KUKA KRL program: EPS_2_25862_MH5A_A_20251016034302.src

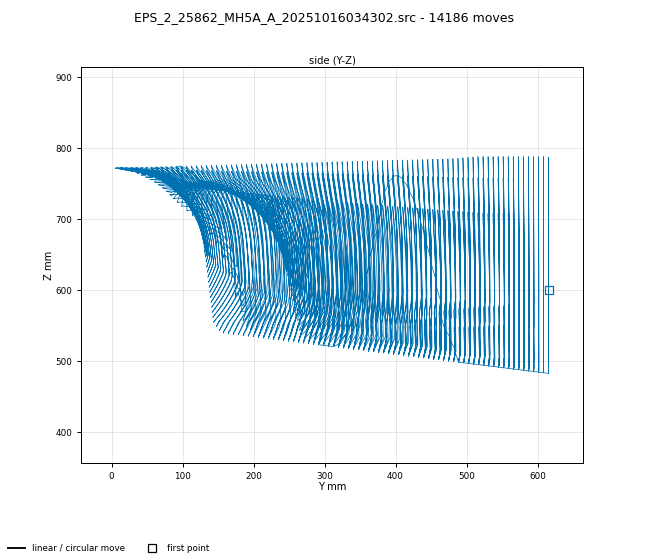
[picture p0: tool path of EPS_2_25862_MH5A_A_20251016034302.src, 14186 of 14188 moves have a stored position in this frame; points joined in program order, loops and branches not executed]
&ACCESS RVP
&REL 4
&COMMENT QRS 19112012
&PARAM EDITMASK = *
DEF PART()
EXT BAS (BAS_COMMAND :IN,REAL :IN )
INT I
BAS (#INITMOV,0 )

;KUKA QRS Post kuka4.cps  Date:22-06-2017 !

File_ID=2891

QRS_PRE_INIT()

;Init var - Until changes are made in qrs_pre_init
Outlet_Square_prg=0
Inlet_1_Square_prg=0
Inlet_2_Square_prg=0
Inlet_3_Square_prg=0
Inlet_4_Square_prg=0
Inlet_5_Square_prg=0

Outlet_1={X 0.000, Y 519.160, Z 687.500, B 0.000, E1 0.000 }
Inlet_1={X 0.000, Y 521.300, Z 657.500, B 0.000, E1 178.000 }
Inlet_2={X 0.000, Y 524.870, Z 607.500, B 0.000, E1 254.000 }
Outlet_1_type=201
Inlet_1_type=201
Inlet_2_type=201
;QRS#1=Sidecore dimensions
;QRS#2=200-8" PVC SDR 35
;QRS#3=200-8" PVC SDR 35
;QRS#4=200-8" PVC SDR 35
;QRS#5=
;QRS#6=
;QRS#7=
;QRS#8=
;QRS#9=12-08 PSX
;QRS#10=12-08 PSX
;QRS#11=12-08 PSX
;QRS#12=
;QRS#13=
;QRS#14=
;QRS#15=
;QRS#16=1220x127x1067 3,5'
;QRS#17=EPS Height
;QRS#18=788
;QRS#19=*
;QRS#20= UPDATED VERSION 22-06-2017
;QRS#21=*
Outlet_Square=0100
Inlet_1_Square=0100
Inlet_2_Square=0100
Inlet_3_Square=0
Inlet_4_Square=0
Inlet_5_Square=0
Mill_Square=1
Outlet_Square_Prg=204
Inlet_1_Square_prg=204
Inlet_2_Square_prg=204

QRS_INIT()

$ADVANCE=5

; T1
PTP {E1 173.595,E2 173.595}
PTP {X 0,Y 615.502,A -85,B 0,C 180,E1 173.595,E2 173.595,E3 0,E4 0,E5 0,E6 0}
QRS_SPEED_INIT()
LIN {X 0,Y 615.502,Z 600,A -85,B 0,C 180,E1 173.595,E2 173.595,E3 0,E4 0,E5 0,E6 0} C_VEL
LIN {X 0,Y 615.502,Z 492.864,A -85,B 0,C 180,E1 173.595,E2 173.595} C_VEL
LIN {X 0,Y 615.502,Z 484.687,A -85,B 0,C 180,E1 173.595,E2 173.595} C_VEL
LIN {X 0,Y 615.49,Z 482.687,A -85,B 0,C 180,E1 173.408,E2 173.408} C_VEL
LIN {X 0,Y 615.493,Z 482.697,A -85,B 0,C 180,E1 170.801,E2 170.801} C_VEL
LIN {X 0,Y 615.479,Z 482.685,A -85,B 0,C 180,E1 168.139,E2 168.139} C_VEL
LIN {X 0,Y 615.488,Z 482.687,A -85,B 0,C 180,E1 165.451,E2 165.451} C_VEL
LIN {X 0,Y 615.492,Z 482.694,A -85,B 0,C 180,E1 162.729,E2 162.729} C_VEL
LIN {X 0,Y 615.477,Z 482.684,A -85,B 0,C 180,E1 159.967,E2 159.967} C_VEL
LIN {X 0,Y 615.494,Z 482.694,A -85,B 0,C 180,E1 157.155,E2 157.155} C_VEL
LIN {X 0,Y 615.493,Z 482.683,A -85,B 0,C 180,E1 154.284,E2 154.284} C_VEL
LIN {X 0,Y 615.484,Z 482.686,A -85,B 0,C 180,E1 151.548,E2 151.548} C_VEL
LIN {X 0,Y 615.491,Z 482.7,A -85,B 0,C 180,E1 148.911,E2 148.911} C_VEL
LIN {X 0,Y 615.479,Z 482.684,A -85,B 0,C 180,E1 145.977,E2 145.977} C_VEL
LIN {X 0,Y 615.481,Z 482.687,A -85,B 0,C 180,E1 143.574,E2 143.574} C_VEL
LIN {X 0,Y 615.495,Z 482.699,A -85,B 0,C 180,E1 140.935,E2 140.935} C_VEL
LIN {X 0,Y 615.488,Z 482.688,A -85,B 0,C 180,E1 138.526,E2 138.526} C_VEL
LIN {X 0,Y 615.477,Z 482.685,A -85,B 0,C 180,E1 135.849,E2 135.849} C_VEL
LIN {X 0,Y 615.496,Z 482.699,A -85,B 0,C 180,E1 133.048,E2 133.048} C_VEL
LIN {X 0,Y 615.489,Z 482.682,A -85,B 0,C 180,E1 130.089,E2 130.089} C_VEL
LIN {X 0,Y 615.492,Z 482.693,A -85,B 0,C 180,E1 127.241,E2 127.241} C_VEL
LIN {X 0,Y 615.485,Z 482.692,A -85,B 0,C 180,E1 124.7,E2 124.7} C_VEL
LIN {X 0,Y 615.49,Z 482.683,A -85,B 0,C 180,E1 122.33,E2 122.33} C_VEL
LIN {X 0,Y 615.476,Z 482.685,A -85,B 0,C 180,E1 119.792,E2 119.792} C_VEL
LIN {X 0,Y 615.498,Z 482.7,A -85,B 0,C 180,E1 117.046,E2 117.046} C_VEL
LIN {X 0,Y 615.489,Z 482.681,A -85,B 0,C 180,E1 114.007,E2 114.007} C_VEL
LIN {X 0,Y 615.474,Z 482.761,A -85,B 0,C 180,E1 113.697,E2 113.697} C_VEL
LIN {X 0,Y 615.484,Z 502.326,A -85,B 0,C 180,E1 110.905,E2 110.905} C_VEL
LIN {X 0,Y 615.489,Z 522.175,A -85,B 0,C 180,E1 108.117,E2 108.117} C_VEL
LIN {X 0,Y 615.494,Z 543.035,A -85,B 0,C 180,E1 105.225,E2 105.225} C_VEL
LIN {X 0,Y 615.481,Z 545.953,A -85,B 0,C 180,E1 104.824,E2 104.824} C_VEL
LIN {X 0,Y 615.48,Z 654.226,A -85,B 0,C 180,E1 103.537,E2 103.537} C_VEL
LIN {X 0,Y 615.487,Z 667.444,A -85,B 0,C 180,E1 103.243,E2 103.243} C_VEL
LIN {X 0,Y 615.487,Z 680.122,A -85,B 0,C 180,E1 102.823,E2 102.823} C_VEL
LIN {X 0,Y 615.487,Z 692.174,A -85,B 0,C 180,E1 102.279,E2 102.279} C_VEL
LIN {X 0,Y 615.49,Z 703.628,A -85,B 0,C 180,E1 101.61,E2 101.61} C_VEL
LIN {X 0,Y 615.496,Z 713.542,A -85,B 0,C 180,E1 100.889,E2 100.889} C_VEL
LIN {X 0,Y 615.497,Z 723.159,A -85,B 0,C 180,E1 100.028,E2 100.028} C_VEL
LIN {X 0,Y 615.496,Z 732.094,A -85,B 0,C 180,E1 99.033,E2 99.033} C_VEL
LIN {X 0,Y 615.499,Z 739.271,A -85,B 0,C 180,E1 98.04,E2 98.04} C_VEL
LIN {X 0,Y 615.496,Z 745.724,A -85,B 0,C 180,E1 96.898,E2 96.898} C_VEL
LIN {X 0,Y 615.497,Z 750.085,A -85,B 0,C 180,E1 95.898,E2 95.898} C_VEL
LIN {X 0,Y 615.498,Z 752.356,A -85,B 0,C 180,E1 95.241,E2 95.241} C_VEL
LIN {X 0,Y 615.496,Z 754.203,A -85,B 0,C 180,E1 94.584,E2 94.584} C_VEL
LIN {X 0,Y 615.496,Z 755.591,A -85,B 0,C 180,E1 93.928,E2 93.928} C_VEL
LIN {X 0,Y 615.495,Z 757.168,A -85,B 0,C 180,E1 92.618,E2 92.618} C_VEL
LIN {X 0,Y 615.5,Z 757.387,A -85,B 0,C 180,E1 91.963,E2 91.963} C_VEL
LIN {X 0,Y 615.495,Z 756.589,A -85,B 0,C 180,E1 90.654,E2 90.654} C_VEL
LIN {X 0,Y 615.497,Z 755.622,A -85,B 0,C 180,E1 90,E2 90} C_VEL
LIN {X 0,Y 615.494,Z 754.255,A -85,B 0,C 180,E1 89.346,E2 89.346} C_VEL
LIN {X 0,Y 615.496,Z 751.382,A -85,B 0,C 180,E1 88.364,E2 88.364} C_VEL
LIN {X 0,Y 615.498,Z 747.492,A -85,B 0,C 180,E1 87.382,E2 87.382} C_VEL
LIN {X 0,Y 615.495,Z 742.483,A -85,B 0,C 180,E1 86.399,E2 86.399} C_VEL
LIN {X 0,Y 615.498,Z 736.194,A -85,B 0,C 180,E1 85.416,E2 85.416} C_VEL
LIN {X 0,Y 615.498,Z 728.32,A -85,B 0,C 180,E1 84.43,E2 84.43} C_VEL
LIN {X 0,Y 615.498,Z 718.54,A -85,B 0,C 180,E1 83.444,E2 83.444} C_VEL
LIN {X 0,Y 615.499,Z 708.271,A -85,B 0,C 180,E1 82.62,E2 82.62} C_VEL
LIN {X 0,Y 615.492,Z 696.728,A -85,B 0,C 180,E1 81.877,E2 81.877} C_VEL
LIN {X 0,Y 615.49,Z 685.198,A -85,B 0,C 180,E1 81.298,E2 81.298} C_VEL
LIN {X 0,Y 615.485,Z 673.274,A -85,B 0,C 180,E1 80.843,E2 80.843} C_VEL
LIN {X 0,Y 615.477,Z 661.229,A -85,B 0,C 180,E1 80.511,E2 80.511} C_VEL
LIN {X 0,Y 615.478,Z 648.035,A -85,B 0,C 180,E1 80.283,E2 80.283} C_VEL
LIN {X 0,Y 615.488,Z 545.884,A -85,B 0,C 180,E1 79.077,E2 79.077} C_VEL
LIN {X 0,Y 615.485,Z 525.776,A -85,B 0,C 180,E1 76.295,E2 76.295} C_VEL
LIN {X 0,Y 615.49,Z 506.326,A -85,B 0,C 180,E1 73.57,E2 73.57} C_VEL
LIN {X 0,Y 615.492,Z 487.095,A -85,B 0,C 180,E1 70.836,E2 70.836} C_VEL
LIN {X 0,Y 615.48,Z 482.686,A -85,B 0,C 180,E1 70.185,E2 70.185} C_VEL
LIN {X 0,Y 615.481,Z 482.685,A -85,B 0,C 180,E1 67.657,E2 67.657} C_VEL
LIN {X 0,Y 615.495,Z 482.699,A -85,B 0,C 180,E1 65.009,E2 65.009} C_VEL
LIN {X 0,Y 615.483,Z 482.683,A -85,B 0,C 180,E1 62.085,E2 62.085} C_VEL
LIN {X 0,Y 615.499,Z 482.68,A -85,B 0,C 180,E1 59.841,E2 59.841} C_VEL
LIN {X 0,Y 615.487,Z 482.687,A -85,B 0,C 180,E1 57.543,E2 57.543} C_VEL
LIN {X 0,Y 615.491,Z 482.697,A -85,B 0,C 180,E1 55.186,E2 55.186} C_VEL
LIN {X 0,Y 615.492,Z 482.691,A -85,B 0,C 180,E1 52.759,E2 52.759} C_VEL
LIN {X 0,Y 615.489,Z 482.682,A -85,B 0,C 180,E1 49.911,E2 49.911} C_VEL
LIN {X 0,Y 615.497,Z 482.694,A -85,B 0,C 180,E1 46.952,E2 46.952} C_VEL
LIN {X 0,Y 615.482,Z 482.684,A -85,B 0,C 180,E1 43.998,E2 43.998} C_VEL
LIN {X 0,Y 615.486,Z 482.7,A -85,B 0,C 180,E1 41.096,E2 41.096} C_VEL
LIN {X 0,Y 615.483,Z 482.693,A -85,B 0,C 180,E1 38.905,E2 38.905} C_VEL
LIN {X 0,Y 615.481,Z 482.684,A -85,B 0,C 180,E1 36.426,E2 36.426} C_VEL
LIN {X 0,Y 615.495,Z 482.691,A -85,B 0,C 180,E1 33.537,E2 33.537} C_VEL
LIN {X 0,Y 615.486,Z 482.884,A -85,B 0,C 180,E1 31.766,E2 31.766} C_VEL
LIN {X 0,Y 615.492,Z 496.948,A -85,B 0,C 180,E1 29.032,E2 29.032} C_VEL
LIN {X 0,Y 615.497,Z 498.159,A -85,B 0,C 180,E1 28.798,E2 28.798} C_VEL
LIN {X 0,Y 615.491,Z 603.751,A -85,B 0,C 180,E1 27.546,E2 27.546} C_VEL
LIN {X 0,Y 615.479,Z 616.47,A -85,B 0,C 180,E1 27.27,E2 27.27} C_VEL
LIN {X 0,Y 615.488,Z 629.197,A -85,B 0,C 180,E1 26.858,E2 26.858} C_VEL
LIN {X 0,Y 615.481,Z 640.719,A -85,B 0,C 180,E1 26.353,E2 26.353} C_VEL
LIN {X 0,Y 615.493,Z 652.002,A -85,B 0,C 180,E1 25.716,E2 25.716} C_VEL
LIN {X 0,Y 615.499,Z 663.389,A -85,B 0,C 180,E1 24.901,E2 24.901} C_VEL
LIN {X 0,Y 615.499,Z 672.008,A -85,B 0,C 180,E1 24.142,E2 24.142} C_VEL
LIN {X 0,Y 615.497,Z 680.725,A -85,B 0,C 180,E1 23.2,E2 23.2} C_VEL
LIN {X 0,Y 615.496,Z 688.627,A -85,B 0,C 180,E1 22.136,E2 22.136} C_VEL
LIN {X 0,Y 615.497,Z 694.828,A -85,B 0,C 180,E1 21.081,E2 21.081} C_VEL
LIN {X 0,Y 615.495,Z 699.584,A -85,B 0,C 180,E1 20.033,E2 20.033} C_VEL
LIN {X 0,Y 615.496,Z 702.046,A -85,B 0,C 180,E1 19.338,E2 19.338} C_VEL
LIN {X 0,Y 615.496,Z 704.133,A -85,B 0,C 180,E1 18.611,E2 18.611} C_VEL
LIN {X 0,Y 615.495,Z 705.544,A -85,B 0,C 180,E1 17.957,E2 17.957} C_VEL
LIN {X 0,Y 615.496,Z 706.572,A -85,B 0,C 180,E1 17.271,E2 17.271} C_VEL
LIN {X 0,Y 615.496,Z 707.28,A -85,B 0,C 180,E1 16.438,E2 16.438} C_VEL
LIN {X 0,Y 615.497,Z 707.12,A -85,B 0,C 180,E1 15.226,E2 15.226} C_VEL
LIN {X 0,Y 615.497,Z 705.525,A -85,B 0,C 180,E1 13.942,E2 13.942} C_VEL
LIN {X 0,Y 615.495,Z 703.871,A -85,B 0,C 180,E1 13.201,E2 13.201} C_VEL
LIN {X 0,Y 615.495,Z 700.772,A -85,B 0,C 180,E1 12.195,E2 12.195} C_VEL
LIN {X 0,Y 615.497,Z 696.609,A -85,B 0,C 180,E1 11.193,E2 11.193} C_VEL
LIN {X 0,Y 615.495,Z 690.251,A -85,B 0,C 180,E1 10.028,E2 10.028} C_VEL
LIN {X 0,Y 615.496,Z 683.344,A -85,B 0,C 180,E1 9.033,E2 9.033} C_VEL
LIN {X 0,Y 615.499,Z 674.712,A -85,B 0,C 180,E1 8.041,E2 8.041} C_VEL
LIN {X 0,Y 615.497,Z 665.894,A -85,B 0,C 180,E1 7.216,E2 7.216} C_VEL
LIN {X 0,Y 615.495,Z 656.246,A -85,B 0,C 180,E1 6.474,E2 6.474} C_VEL
LIN {X 0,Y 615.481,Z 645.657,A -85,B 0,C 180,E1 5.817,E2 5.817} C_VEL
LIN {X 0,Y 615.495,Z 633.852,A -85,B 0,C 180,E1 5.241,E2 5.241} C_VEL
LIN {X 0,Y 615.483,Z 621.635,A -85,B 0,C 180,E1 4.79,E2 4.79} C_VEL
LIN {X 0,Y 615.492,Z 609.025,A -85,B 0,C 180,E1 4.462,E2 4.462} C_VEL
LIN {X 0,Y 615.493,Z 593.991,A -85,B 0,C 180,E1 4.236,E2 4.236} C_VEL
LIN {X 0,Y 615.487,Z 498.146,A -85,B 0,C 180,E1 3.109,E2 3.109} C_VEL
LIN {X 0,Y 615.487,Z 483.823,A -85,B 0,C 180,E1 0.327,E2 0.327} C_VEL
LIN {X 0,Y 615.477,Z 482.689,A -85,B 0,C 180,E1 0.082,E2 0.082} C_VEL
LIN {X 0,Y 615.493,Z 482.682,A -85,B 0,C 180,E1 -2.618,E2 -2.618} C_VEL
LIN {X 0,Y 615.495,Z 482.698,A -85,B 0,C 180,E1 -5.241,E2 -5.241} C_VEL
LIN {X 0,Y 615.479,Z 482.688,A -85,B 0,C 180,E1 -7.876,E2 -7.876} C_VEL
LIN {X 0,Y 615.49,Z 482.683,A -85,B 0,C 180,E1 -10.527,E2 -10.527} C_VEL
LIN {X 0,Y 615.497,Z 482.699,A -85,B 0,C 180,E1 -13.201,E2 -13.201} C_VEL
LIN {X 0,Y 615.48,Z 482.686,A -85,B 0,C 180,E1 -15.905,E2 -15.905} C_VEL
LIN {X 0,Y 615.492,Z 482.685,A -85,B 0,C 180,E1 -18.646,E2 -18.646} C_VEL
LIN {X 0,Y 615.495,Z 482.692,A -85,B 0,C 180,E1 -21.432,E2 -21.432} C_VEL
LIN {X 0,Y 615.478,Z 482.685,A -85,B 0,C 180,E1 -24.272,E2 -24.272} C_VEL
LIN {X 0,Y 615.497,Z 482.698,A -85,B 0,C 180,E1 -27.049,E2 -27.049} C_VEL
LIN {X 0,Y 615.488,Z 482.684,A -85,B 0,C 180,E1 -29.797,E2 -29.797} C_VEL
LIN {X 0,Y 615.484,Z 482.686,A -85,B 0,C 180,E1 -32.458,E2 -32.458} C_VEL
LIN {X 0,Y 615.497,Z 482.692,A -85,B 0,C 180,E1 -34.815,E2 -34.815} C_VEL
LIN {X 0,Y 615.482,Z 482.697,A -85,B 0,C 180,E1 -37.243,E2 -37.243} C_VEL
LIN {X 0,Y 615.498,Z 482.681,A -85,B 0,C 180,E1 -39.749,E2 -39.749} C_VEL
LIN {X 0,Y 615.474,Z 482.688,A -85,B 0,C 180,E1 -42.354,E2 -42.354} C_VEL
LIN {X 0,Y 615.492,Z 482.698,A -85,B 0,C 180,E1 -45.068,E2 -45.068} C_VEL
LIN {X 0,Y 615.488,Z 482.682,A -85,B 0,C 180,E1 -47.92,E2 -47.92} C_VEL
LIN {X 0,Y 615.477,Z 482.687,A -85,B 0,C 180,E1 -50.25,E2 -50.25} C_VEL
LIN {X 0,Y 615.484,Z 482.697,A -85,B 0,C 180,E1 -53.064,E2 -53.064} C_VEL
LIN {X 0,Y 615.487,Z 482.682,A -85,B 0,C 180,E1 -55.979,E2 -55.979} C_VEL
LIN {X 0,Y 615.488,Z 482.7,A -85,B 0,C 180,E1 -58.914,E2 -58.914} C_VEL
LIN {X 0,Y 615.48,Z 482.685,A -85,B 0,C 180,E1 -61.551,E2 -61.551} C_VEL
LIN {X 0,Y 615.477,Z 482.689,A -85,B 0,C 180,E1 -64.284,E2 -64.284} C_VEL
LIN {X 0,Y 615.488,Z 482.751,A -85,B 0,C 180,E1 -66.02,E2 -66.02} C_VEL
LIN {X 0,Y 615.496,Z 506.248,A -85,B 0,C 180,E1 -68.92,E2 -68.92} C_VEL
LIN {X 0,Y 615.483,Z 530.707,A -85,B 0,C 180,E1 -71.881,E2 -71.881} C_VEL
LIN {X 0,Y 615.498,Z 554.974,A -85,B 0,C 180,E1 -74.775,E2 -74.775} C_VEL
LIN {X 0,Y 615.49,Z 574.818,A -85,B 0,C 180,E1 -77.114,E2 -77.114} C_VEL
LIN {X 0,Y 615.477,Z 683.848,A -85,B 0,C 180,E1 -78.411,E2 -78.411} C_VEL
LIN {X 0,Y 615.482,Z 696.355,A -85,B 0,C 180,E1 -78.682,E2 -78.682} C_VEL
LIN {X 0,Y 615.497,Z 709.489,A -85,B 0,C 180,E1 -79.108,E2 -79.108} C_VEL
LIN {X 0,Y 615.48,Z 721.483,A -85,B 0,C 180,E1 -79.64,E2 -79.64} C_VEL
LIN {X 0,Y 615.481,Z 733,A -85,B 0,C 180,E1 -80.304,E2 -80.304} C_VEL
LIN {X 0,Y 615.499,Z 743.344,A -85,B 0,C 180,E1 -81.05,E2 -81.05} C_VEL
LIN {X 0,Y 615.497,Z 751.814,A -85,B 0,C 180,E1 -81.794,E2 -81.794} C_VEL
LIN {X 0,Y 615.498,Z 759.608,A -85,B 0,C 180,E1 -82.62,E2 -82.62} C_VEL
LIN {X 0,Y 615.496,Z 767.204,A -85,B 0,C 180,E1 -83.608,E2 -83.608} C_VEL
LIN {X 0,Y 615.498,Z 774.205,A -85,B 0,C 180,E1 -84.759,E2 -84.759} C_VEL
LIN {X 0,Y 615.493,Z 778.852,A -85,B 0,C 180,E1 -85.744,E2 -85.744} C_VEL
LIN {X 0,Y 615.495,Z 782.399,A -85,B 0,C 180,E1 -86.727,E2 -86.727} C_VEL
LIN {X 0,Y 615.497,Z 784.233,A -85,B 0,C 180,E1 -87.382,E2 -87.382} C_VEL
LIN {X 0,Y 615.496,Z 785.608,A -85,B 0,C 180,E1 -88.037,E2 -88.037} C_VEL
LIN {X 0,Y 615.496,Z 787.174,A -85,B 0,C 180,E1 -89.346,E2 -89.346} C_VEL
LIN {X 0,Y 615.494,Z 787.389,A -85,B 0,C 180,E1 -90,E2 -90} C_VEL
LIN {X 0,Y 615.496,Z 786.58,A -85,B 0,C 180,E1 -91.309,E2 -91.309} C_VEL
LIN {X 0,Y 615.496,Z 785.608,A -85,B 0,C 180,E1 -91.963,E2 -91.963} C_VEL
LIN {X 0,Y 615.497,Z 784.233,A -85,B 0,C 180,E1 -92.618,E2 -92.618} C_VEL
LIN {X 0,Y 615.496,Z 781.35,A -85,B 0,C 180,E1 -93.601,E2 -93.601} C_VEL
LIN {X 0,Y 615.498,Z 777.442,A -85,B 0,C 180,E1 -94.584,E2 -94.584} C_VEL
LIN {X 0,Y 615.499,Z 772.406,A -85,B 0,C 180,E1 -95.57,E2 -95.57} C_VEL
LIN {X 0,Y 615.497,Z 765.869,A -85,B 0,C 180,E1 -96.583,E2 -96.583} C_VEL
LIN {X 0,Y 615.497,Z 758.135,A -85,B 0,C 180,E1 -97.545,E2 -97.545} C_VEL
LIN {X 0,Y 615.498,Z 750.047,A -85,B 0,C 180,E1 -98.371,E2 -98.371} C_VEL
LIN {X 0,Y 615.499,Z 740.17,A -85,B 0,C 180,E1 -99.198,E2 -99.198} C_VEL
LIN {X 0,Y 615.483,Z 728.986,A -85,B 0,C 180,E1 -99.945,E2 -99.945} C_VEL
LIN {X 0,Y 615.481,Z 718.029,A -85,B 0,C 180,E1 -100.527,E2 -100.527} C_VEL
LIN {X 0,Y 615.499,Z 705.423,A -85,B 0,C 180,E1 -101.042,E2 -101.042} C_VEL
LIN {X 0,Y 615.479,Z 693.079,A -85,B 0,C 180,E1 -101.401,E2 -101.401} C_VEL
LIN {X 0,Y 615.477,Z 679.489,A -85,B 0,C 180,E1 -101.652,E2 -101.652} C_VEL
LIN {X 0,Y 615.49,Z 574.818,A -85,B 0,C 180,E1 -102.886,E2 -102.886} C_VEL
LIN {X 0,Y 615.479,Z 550.678,A -85,B 0,C 180,E1 -105.735,E2 -105.735} C_VEL
LIN {X 0,Y 615.493,Z 528.001,A -85,B 0,C 180,E1 -108.444,E2 -108.444} C_VEL
LIN {X 0,Y 615.495,Z 504.813,A -85,B 0,C 180,E1 -111.255,E2 -111.255} C_VEL
LIN {X 0,Y 615.489,Z 482.683,A -85,B 0,C 180,E1 -113.994,E2 -113.994} C_VEL
LIN {X 0,Y 615.48,Z 482.685,A -85,B 0,C 180,E1 -116.444,E2 -116.444} C_VEL
LIN {X 0,Y 615.477,Z 482.689,A -85,B 0,C 180,E1 -118.658,E2 -118.658} C_VEL
LIN {X 0,Y 615.489,Z 482.698,A -85,B 0,C 180,E1 -121.086,E2 -121.086} C_VEL
LIN {X 0,Y 615.487,Z 482.683,A -85,B 0,C 180,E1 -124.021,E2 -124.021} C_VEL
LIN {X 0,Y 615.482,Z 482.695,A -85,B 0,C 180,E1 -126.936,E2 -126.936} C_VEL
LIN {X 0,Y 615.477,Z 482.688,A -85,B 0,C 180,E1 -129.75,E2 -129.75} C_VEL
LIN {X 0,Y 615.49,Z 482.682,A -85,B 0,C 180,E1 -132.351,E2 -132.351} C_VEL
LIN {X 0,Y 615.48,Z 482.7,A -85,B 0,C 180,E1 -135.068,E2 -135.068} C_VEL
LIN {X 0,Y 615.477,Z 482.686,A -85,B 0,C 180,E1 -137.919,E2 -137.919} C_VEL
LIN {X 0,Y 615.498,Z 482.68,A -85,B 0,C 180,E1 -140.251,E2 -140.251} C_VEL
LIN {X 0,Y 615.478,Z 482.701,A -85,B 0,C 180,E1 -143.063,E2 -143.063} C_VEL
LIN {X 0,Y 615.495,Z 482.696,A -85,B 0,C 180,E1 -145.296,E2 -145.296} C_VEL
LIN {X 0,Y 615.485,Z 482.683,A -85,B 0,C 180,E1 -148.314,E2 -148.314} C_VEL
LIN {X 0,Y 615.482,Z 482.687,A -85,B 0,C 180,E1 -150.593,E2 -150.593} C_VEL
LIN {X 0,Y 615.479,Z 482.698,A -85,B 0,C 180,E1 -152.954,E2 -152.954} C_VEL
LIN {X 0,Y 615.478,Z 482.688,A -85,B 0,C 180,E1 -155.728,E2 -155.728} C_VEL
LIN {X 0,Y 615.486,Z 482.686,A -85,B 0,C 180,E1 -158.568,E2 -158.568} C_VEL
LIN {X 0,Y 615.495,Z 482.692,A -85,B 0,C 180,E1 -161.389,E2 -161.389} C_VEL
LIN {X 0,Y 615.48,Z 482.684,A -85,B 0,C 180,E1 -164.095,E2 -164.095} C_VEL
LIN {X 0,Y 615.479,Z 482.693,A -85,B 0,C 180,E1 -166.799,E2 -166.799} C_VEL
LIN {X 0,Y 615.491,Z 482.69,A -85,B 0,C 180,E1 -169.473,E2 -169.473} C_VEL
LIN {X 0,Y 615.479,Z 482.684,A -85,B 0,C 180,E1 -172.124,E2 -172.124} C_VEL
LIN {X 0,Y 615.483,Z 482.692,A -85,B 0,C 180,E1 -174.759,E2 -174.759} C_VEL
LIN {X 0,Y 615.497,Z 482.691,A -85,B 0,C 180,E1 -177.382,E2 -177.382} C_VEL
LIN {X 0,Y 615.477,Z 482.685,A -85,B 0,C 180,E1 -180,E2 -180} C_VEL
LIN {X 0,Y 615.491,Z 482.687,A -85,B 0,C 180,E1 -182.618,E2 -182.618} C_VEL
LIN {X 0,Y 615.493,Z 482.696,A -85,B 0,C 180,E1 -185.241,E2 -185.241} C_VEL
LIN {X 0,Y 615.49,Z 482.687,A -85,B 0,C 180,E1 -186.592,E2 -186.592} C_VEL
LIN {X 0,Y 614.816,Z 482.842,A -85,B 0,C 180,E1 -187.138,E2 -187.138} C_VEL
LIN {X 0,Y 611.984,Z 483.247,A -85,B 0,C 180,E1 -188.024,E2 -188.024} C_VEL
LIN {X 0,Y 609.59,Z 483.561,A -85,B 0,C 180,E1 -188.736,E2 -188.736} C_VEL
LIN {X 0,Y 608.55,Z 483.682,A -85,B 0,C 180,E1 -189.286,E2 -189.286} C_VEL
LIN {X 0,Y 608.459,Z 483.69,A -85,B 0,C 180,E1 -189.472,E2 -189.472} C_VEL
LIN {X 0,Y 608.456,Z 483.687,A -85,B 0,C 180,E1 -192,E2 -192} C_VEL
LIN {X 0,Y 608.476,Z 483.689,A -85,B 0,C 180,E1 -194.721,E2 -194.721} C_VEL
LIN {X 0,Y 608.453,Z 483.691,A -85,B 0,C 180,E1 -197.477,E2 -197.477} C_VEL
LIN {X 0,Y 608.459,Z 483.687,A -85,B 0,C 180,E1 -200.275,E2 -200.275} C_VEL
LIN {X 0,Y 608.455,Z 483.696,A -85,B 0,C 180,E1 -203.124,E2 -203.124} C_VEL
LIN {X 0,Y 608.448,Z 483.688,A -85,B 0,C 180,E1 -206.036,E2 -206.036} C_VEL
LIN {X 0,Y 608.473,Z 483.688,A -85,B 0,C 180,E1 -208.622,E2 -208.622} C_VEL
LIN {X 0,Y 608.474,Z 483.69,A -85,B 0,C 180,E1 -211.316,E2 -211.316} C_VEL
LIN {X 0,Y 608.472,Z 483.686,A -85,B 0,C 180,E1 -213.737,E2 -213.737} C_VEL
LIN {X 0,Y 608.472,Z 483.685,A -85,B 0,C 180,E1 -216.091,E2 -216.091} C_VEL
LIN {X 0,Y 608.472,Z 483.688,A -85,B 0,C 180,E1 -218.588,E2 -218.588} C_VEL
LIN {X 0,Y 608.466,Z 483.691,A -85,B 0,C 180,E1 -221.344,E2 -221.344} C_VEL
LIN {X 0,Y 608.449,Z 483.688,A -85,B 0,C 180,E1 -224.265,E2 -224.265} C_VEL
LIN {X 0,Y 608.462,Z 483.697,A -85,B 0,C 180,E1 -227.042,E2 -227.042} C_VEL
LIN {X 0,Y 608.454,Z 483.688,A -85,B 0,C 180,E1 -229.698,E2 -229.698} C_VEL
LIN {X 0,Y 608.47,Z 483.686,A -85,B 0,C 180,E1 -232.255,E2 -232.255} C_VEL
LIN {X 0,Y 608.452,Z 483.696,A -85,B 0,C 180,E1 -235.095,E2 -235.095} C_VEL
LIN {X 0,Y 608.467,Z 483.685,A -85,B 0,C 180,E1 -237.906,E2 -237.906} C_VEL
LIN {X 0,Y 608.462,Z 483.687,A -85,B 0,C 180,E1 -240.221,E2 -240.221} C_VEL
LIN {X 0,Y 608.485,Z 483.691,A -85,B 0,C 180,E1 -242.793,E2 -242.793} C_VEL
LIN {X 0,Y 608.482,Z 483.684,A -85,B 0,C 180,E1 -245.848,E2 -245.848} C_VEL
LIN {X 0,Y 608.486,Z 483.874,A -85,B 0,C 180,E1 -246.202,E2 -246.202} C_VEL
LIN {X 0,Y 608.541,Z 502.176,A -85,B 0,C 180,E1 -248.845,E2 -248.845} C_VEL
LIN {X 0,Y 608.516,Z 522.072,A -85,B 0,C 180,E1 -251.668,E2 -251.668} C_VEL
LIN {X 0,Y 608.484,Z 543.003,A -85,B 0,C 180,E1 -254.595,E2 -254.595} C_VEL
LIN {X 0,Y 608.468,Z 546.09,A -85,B 0,C 180,E1 -255.023,E2 -255.023} C_VEL
LIN {X 0,Y 608.539,Z 654.234,A -85,B 0,C 180,E1 -256.327,E2 -256.327} C_VEL
LIN {X 0,Y 608.533,Z 667.487,A -85,B 0,C 180,E1 -256.624,E2 -256.624} C_VEL
LIN {X 0,Y 608.513,Z 679.635,A -85,B 0,C 180,E1 -257.027,E2 -257.027} C_VEL
LIN {X 0,Y 608.512,Z 691.904,A -85,B 0,C 180,E1 -257.578,E2 -257.578} C_VEL
LIN {X 0,Y 608.497,Z 703.48,A -85,B 0,C 180,E1 -258.255,E2 -258.255} C_VEL
LIN {X 0,Y 608.481,Z 714.238,A -85,B 0,C 180,E1 -259.042,E2 -259.042} C_VEL
LIN {X 0,Y 608.482,Z 723.247,A -85,B 0,C 180,E1 -259.855,E2 -259.855} C_VEL
LIN {X 0,Y 608.47,Z 732.28,A -85,B 0,C 180,E1 -260.862,E2 -260.862} C_VEL
LIN {X 0,Y 608.464,Z 739.55,A -85,B 0,C 180,E1 -261.866,E2 -261.866} C_VEL
LIN {X 0,Y 608.445,Z 744.449,A -85,B 0,C 180,E1 -262.701,E2 -262.701} C_VEL
LIN {X 0,Y 608.452,Z 748.911,A -85,B 0,C 180,E1 -263.632,E2 -263.632} C_VEL
LIN {X 0,Y 608.442,Z 752.841,A -85,B 0,C 180,E1 -264.698,E2 -264.698} C_VEL
LIN {X 0,Y 608.429,Z 754.719,A -85,B 0,C 180,E1 -265.362,E2 -265.362} C_VEL
LIN {X 0,Y 608.433,Z 756.146,A -85,B 0,C 180,E1 -266.026,E2 -266.026} C_VEL
LIN {X 0,Y 608.421,Z 757.761,A -85,B 0,C 180,E1 -267.352,E2 -267.352} C_VEL
LIN {X 0,Y 608.445,Z 757.998,A -85,B 0,C 180,E1 -268.014,E2 -268.014} C_VEL
LIN {X 0,Y 608.447,Z 757.805,A -85,B 0,C 180,E1 -268.676,E2 -268.676} C_VEL
LIN {X 0,Y 608.437,Z 756.252,A -85,B 0,C 180,E1 -270,E2 -270} C_VEL
LIN {X 0,Y 608.437,Z 754.886,A -85,B 0,C 180,E1 -270.662,E2 -270.662} C_VEL
LIN {X 0,Y 608.44,Z 752.003,A -85,B 0,C 180,E1 -271.655,E2 -271.655} C_VEL
LIN {X 0,Y 608.432,Z 748.099,A -85,B 0,C 180,E1 -272.648,E2 -272.648} C_VEL
LIN {X 0,Y 608.449,Z 743.07,A -85,B 0,C 180,E1 -273.642,E2 -273.642} C_VEL
LIN {X 0,Y 608.465,Z 736.761,A -85,B 0,C 180,E1 -274.637,E2 -274.637} C_VEL
LIN {X 0,Y 608.47,Z 728.87,A -85,B 0,C 180,E1 -275.634,E2 -275.634} C_VEL
LIN {X 0,Y 608.485,Z 719.072,A -85,B 0,C 180,E1 -276.632,E2 -276.632} C_VEL
LIN {X 0,Y 608.479,Z 708.818,A -85,B 0,C 180,E1 -277.466,E2 -277.466} C_VEL
LIN {X 0,Y 608.507,Z 697.295,A -85,B 0,C 180,E1 -278.217,E2 -278.217} C_VEL
LIN {X 0,Y 608.511,Z 685.877,A -85,B 0,C 180,E1 -278.802,E2 -278.802} C_VEL
LIN {X 0,Y 608.533,Z 674.107,A -85,B 0,C 180,E1 -279.263,E2 -279.263} C_VEL
LIN {X 0,Y 608.518,Z 660.533,A -85,B 0,C 180,E1 -279.64,E2 -279.64} C_VEL
LIN {X 0,Y 608.552,Z 648.33,A -85,B 0,C 180,E1 -279.85,E2 -279.85} C_VEL
LIN {X 0,Y 608.476,Z 546.03,A -85,B 0,C 180,E1 -281.075,E2 -281.075} C_VEL
LIN {X 0,Y 608.5,Z 525.828,A -85,B 0,C 180,E1 -283.894,E2 -283.894} C_VEL
LIN {X 0,Y 608.511,Z 507.114,A -85,B 0,C 180,E1 -286.541,E2 -286.541} C_VEL
LIN {X 0,Y 608.556,Z 488.485,A -85,B 0,C 180,E1 -289.216,E2 -289.216} C_VEL
LIN {X 0,Y 608.457,Z 483.689,A -85,B 0,C 180,E1 -289.921,E2 -289.921} C_VEL
LIN {X 0,Y 608.463,Z 483.688,A -85,B 0,C 180,E1 -292.476,E2 -292.476} C_VEL
LIN {X 0,Y 608.458,Z 483.69,A -85,B 0,C 180,E1 -294.57,E2 -294.57} C_VEL
LIN {X 0,Y 608.486,Z 483.691,A -85,B 0,C 180,E1 -297.207,E2 -297.207} C_VEL
LIN {X 0,Y 608.465,Z 483.686,A -85,B 0,C 180,E1 -299.97,E2 -299.97} C_VEL
LIN {X 0,Y 608.462,Z 483.689,A -85,B 0,C 180,E1 -302.522,E2 -302.522} C_VEL
LIN {X 0,Y 608.439,Z 483.694,A -85,B 0,C 180,E1 -305.277,E2 -305.277} C_VEL
LIN {X 0,Y 608.47,Z 483.685,A -85,B 0,C 180,E1 -307.745,E2 -307.745} C_VEL
LIN {X 0,Y 608.455,Z 483.689,A -85,B 0,C 180,E1 -310.329,E2 -310.329} C_VEL
LIN {X 0,Y 608.485,Z 483.687,A -85,B 0,C 180,E1 -313.31,E2 -313.31} C_VEL
LIN {X 0,Y 608.469,Z 483.686,A -85,B 0,C 180,E1 -316.13,E2 -316.13} C_VEL
LIN {X 0,Y 608.457,Z 483.698,A -85,B 0,C 180,E1 -318.823,E2 -318.823} C_VEL
LIN {X 0,Y 608.465,Z 483.687,A -85,B 0,C 180,E1 -321.411,E2 -321.411} C_VEL
LIN {X 0,Y 608.472,Z 483.685,A -85,B 0,C 180,E1 -323.949,E2 -323.949} C_VEL
LIN {X 0,Y 608.467,Z 483.689,A -85,B 0,C 180,E1 -326.329,E2 -326.329} C_VEL
LIN {X 0,Y 608.47,Z 483.805,A -85,B 0,C 180,E1 -328.198,E2 -328.198} C_VEL
LIN {X 0,Y 608.469,Z 498.316,A -85,B 0,C 180,E1 -331.038,E2 -331.038} C_VEL
LIN {X 0,Y 608.588,Z 508.378,A -85,B 0,C 180,E1 -331.176,E2 -331.176} C_VEL
LIN {X 0,Y 608.538,Z 604.65,A -85,B 0,C 180,E1 -332.334,E2 -332.334} C_VEL
LIN {X 0,Y 608.519,Z 618.171,A -85,B 0,C 180,E1 -332.643,E2 -332.643} C_VEL
LIN {X 0,Y 608.526,Z 630.922,A -85,B 0,C 180,E1 -333.077,E2 -333.077} C_VEL
LIN {X 0,Y 608.506,Z 642.266,A -85,B 0,C 180,E1 -333.598,E2 -333.598} C_VEL
LIN {X 0,Y 608.481,Z 653.778,A -85,B 0,C 180,E1 -334.274,E2 -334.274} C_VEL
LIN {X 0,Y 608.483,Z 664.536,A -85,B 0,C 180,E1 -335.066,E2 -335.066} C_VEL
LIN {X 0,Y 608.465,Z 674.673,A -85,B 0,C 180,E1 -336.002,E2 -336.002} C_VEL
LIN {X 0,Y 608.469,Z 682.396,A -85,B 0,C 180,E1 -336.876,E2 -336.876} C_VEL
LIN {X 0,Y 608.454,Z 690.095,A -85,B 0,C 180,E1 -337.951,E2 -337.951} C_VEL
LIN {X 0,Y 608.431,Z 696.085,A -85,B 0,C 180,E1 -339.017,E2 -339.017} C_VEL
LIN {X 0,Y 608.434,Z 700.699,A -85,B 0,C 180,E1 -340.077,E2 -340.077} C_VEL
LIN {X 0,Y 608.425,Z 704.533,A -85,B 0,C 180,E1 -341.293,E2 -341.293} C_VEL
LIN {X 0,Y 608.42,Z 706.949,A -85,B 0,C 180,E1 -342.522,E2 -342.522} C_VEL
LIN {X 0,Y 608.422,Z 707.851,A -85,B 0,C 180,E1 -343.481,E2 -343.481} C_VEL
LIN {X 0,Y 608.42,Z 707.863,A -85,B 0,C 180,E1 -344.592,E2 -344.592} C_VEL
LIN {X 0,Y 608.418,Z 707.29,A -85,B 0,C 180,E1 -345.278,E2 -345.278} C_VEL
LIN {X 0,Y 608.431,Z 706.267,A -85,B 0,C 180,E1 -345.992,E2 -345.992} C_VEL
LIN {X 0,Y 608.437,Z 704.93,A -85,B 0,C 180,E1 -346.643,E2 -346.643} C_VEL
LIN {X 0,Y 608.431,Z 701.982,A -85,B 0,C 180,E1 -347.661,E2 -347.661} C_VEL
LIN {X 0,Y 608.452,Z 697.98,A -85,B 0,C 180,E1 -348.676,E2 -348.676} C_VEL
LIN {X 0,Y 608.443,Z 691.825,A -85,B 0,C 180,E1 -349.854,E2 -349.854} C_VEL
LIN {X 0,Y 608.469,Z 685.104,A -85,B 0,C 180,E1 -350.862,E2 -350.862} C_VEL
LIN {X 0,Y 608.462,Z 676.803,A -85,B 0,C 180,E1 -351.866,E2 -351.866} C_VEL
LIN {X 0,Y 608.49,Z 668.305,A -85,B 0,C 180,E1 -352.701,E2 -352.701} C_VEL
LIN {X 0,Y 608.476,Z 657.879,A -85,B 0,C 180,E1 -353.534,E2 -353.534} C_VEL
LIN {X 0,Y 608.483,Z 647.596,A -85,B 0,C 180,E1 -354.199,E2 -354.199} C_VEL
LIN {X 0,Y 608.526,Z 636.324,A -85,B 0,C 180,E1 -354.782,E2 -354.782} C_VEL
LIN {X 0,Y 608.526,Z 624.862,A -85,B 0,C 180,E1 -355.238,E2 -355.238} C_VEL
LIN {X 0,Y 608.55,Z 611.74,A -85,B 0,C 180,E1 -355.612,E2 -355.612} C_VEL
LIN {X 0,Y 608.552,Z 599.021,A -85,B 0,C 180,E1 -355.84,E2 -355.84} C_VEL
LIN {X 0,Y 608.449,Z 498.372,A -85,B 0,C 180,E1 -357.041,E2 -357.041} C_VEL
LIN {X 0,Y 608.451,Z 484.1,A -85,B 0,C 180,E1 -359.834,E2 -359.834} C_VEL
LIN {X 0,Y 608.467,Z 483.687,A -85,B 0,C 180,E1 -360,E2 -360} C_VEL
LIN {X 0,Y 608.482,Z 483.685,A -85,B 0,C 180,E1 -362.648,E2 -362.648} C_VEL
LIN {X 0,Y 608.471,Z 483.696,A -85,B 0,C 180,E1 -365.302,E2 -365.302} C_VEL
LIN {X 0,Y 608.471,Z 483.686,A -85,B 0,C 180,E1 -367.967,E2 -367.967} C_VEL
LIN {X 0,Y 608.467,Z 483.687,A -85,B 0,C 180,E1 -370.65,E2 -370.65} C_VEL
LIN {X 0,Y 608.469,Z 483.694,A -85,B 0,C 180,E1 -373.356,E2 -373.356} C_VEL
LIN {X 0,Y 608.455,Z 483.687,A -85,B 0,C 180,E1 -376.094,E2 -376.094} C_VEL
LIN {X 0,Y 608.456,Z 483.692,A -85,B 0,C 180,E1 -378.87,E2 -378.87} C_VEL
LIN {X 0,Y 608.47,Z 483.688,A -85,B 0,C 180,E1 -381.691,E2 -381.691} C_VEL
LIN {X 0,Y 608.451,Z 483.689,A -85,B 0,C 180,E1 -384.571,E2 -384.571} C_VEL
LIN {X 0,Y 608.482,Z 483.693,A -85,B 0,C 180,E1 -387.211,E2 -387.211} C_VEL
LIN {X 0,Y 608.464,Z 483.686,A -85,B 0,C 180,E1 -389.973,E2 -389.973} C_VEL
LIN {X 0,Y 608.458,Z 483.689,A -85,B 0,C 180,E1 -392.524,E2 -392.524} C_VEL
LIN {X 0,Y 608.453,Z 483.694,A -85,B 0,C 180,E1 -395.277,E2 -395.277} C_VEL
LIN {X 0,Y 608.464,Z 483.687,A -85,B 0,C 180,E1 -397.747,E2 -397.747} C_VEL
LIN {X 0,Y 608.447,Z 483.689,A -85,B 0,C 180,E1 -400.33,E2 -400.33} C_VEL
LIN {X 0,Y 608.465,Z 483.691,A -85,B 0,C 180,E1 -403.31,E2 -403.31} C_VEL
LIN {X 0,Y 608.469,Z 483.686,A -85,B 0,C 180,E1 -406.132,E2 -406.132} C_VEL
LIN {X 0,Y 608.455,Z 483.696,A -85,B 0,C 180,E1 -408.825,E2 -408.825} C_VEL
LIN {X 0,Y 608.466,Z 483.688,A -85,B 0,C 180,E1 -411.413,E2 -411.413} C_VEL
LIN {X 0,Y 608.457,Z 483.687,A -85,B 0,C 180,E1 -413.953,E2 -413.953} C_VEL
LIN {X 0,Y 608.463,Z 483.688,A -85,B 0,C 180,E1 -416.33,E2 -416.33} C_VEL
LIN {X 0,Y 608.476,Z 483.693,A -85,B 0,C 180,E1 -418.728,E2 -418.728} C_VEL
LIN {X 0,Y 608.466,Z 483.688,A -85,B 0,C 180,E1 -421.382,E2 -421.382} C_VEL
LIN {X 0,Y 608.438,Z 483.69,A -85,B 0,C 180,E1 -423.965,E2 -423.965} C_VEL
LIN {X 0,Y 608.482,Z 483.708,A -85,B 0,C 180,E1 -425.847,E2 -425.847} C_VEL
LIN {X 0,Y 608.609,Z 499.073,A -85,B 0,C 180,E1 -427.779,E2 -427.779} C_VEL
LIN {X 0,Y 608.544,Z 522.033,A -85,B 0,C 180,E1 -430.608,E2 -430.608} C_VEL
LIN {X 0,Y 608.525,Z 543.558,A -85,B 0,C 180,E1 -433.218,E2 -433.218} C_VEL
LIN {X 0,Y 608.504,Z 566.578,A -85,B 0,C 180,E1 -435.971,E2 -435.971} C_VEL
LIN {X 0,Y 608.524,Z 575.275,A -85,B 0,C 180,E1 -436.974,E2 -436.974} C_VEL
LIN {X 0,Y 608.534,Z 683.962,A -85,B 0,C 180,E1 -438.277,E2 -438.277} C_VEL
LIN {X 0,Y 608.533,Z 697.225,A -85,B 0,C 180,E1 -438.572,E2 -438.572} C_VEL
LIN {X 0,Y 608.544,Z 710.333,A -85,B 0,C 180,E1 -439.009,E2 -439.009} C_VEL
LIN {X 0,Y 608.498,Z 721.64,A -85,B 0,C 180,E1 -439.519,E2 -439.519} C_VEL
LIN {X 0,Y 608.471,Z 733.201,A -85,B 0,C 180,E1 -440.191,E2 -440.191} C_VEL
LIN {X 0,Y 608.485,Z 743.596,A -85,B 0,C 180,E1 -440.946,E2 -440.946} C_VEL
LIN {X 0,Y 608.475,Z 752.114,A -85,B 0,C 180,E1 -441.699,E2 -441.699} C_VEL
LIN {X 0,Y 608.471,Z 759.962,A -85,B 0,C 180,E1 -442.534,E2 -442.534} C_VEL
LIN {X 0,Y 608.46,Z 767.287,A -85,B 0,C 180,E1 -443.485,E2 -443.485} C_VEL
LIN {X 0,Y 608.45,Z 772.867,A -85,B 0,C 180,E1 -444.366,E2 -444.366} C_VEL
LIN {X 0,Y 608.432,Z 777.951,A -85,B 0,C 180,E1 -445.362,E2 -445.362} C_VEL
LIN {X 0,Y 608.449,Z 781.896,A -85,B 0,C 180,E1 -446.358,E2 -446.358} C_VEL
LIN {X 0,Y 608.425,Z 784.809,A -85,B 0,C 180,E1 -447.352,E2 -447.352} C_VEL
LIN {X 0,Y 608.441,Z 786.201,A -85,B 0,C 180,E1 -448.014,E2 -448.014} C_VEL
LIN {X 0,Y 608.438,Z 787.783,A -85,B 0,C 180,E1 -449.338,E2 -449.338} C_VEL
LIN {X 0,Y 608.434,Z 788,A -85,B 0,C 180,E1 -450,E2 -450} C_VEL
LIN {X 0,Y 608.448,Z 787.184,A -85,B 0,C 180,E1 -451.324,E2 -451.324} C_VEL
LIN {X 0,Y 608.441,Z 786.201,A -85,B 0,C 180,E1 -451.986,E2 -451.986} C_VEL
LIN {X 0,Y 608.425,Z 784.809,A -85,B 0,C 180,E1 -452.648,E2 -452.648} C_VEL
LIN {X 0,Y 608.449,Z 781.896,A -85,B 0,C 180,E1 -453.642,E2 -453.642} C_VEL
LIN {X 0,Y 608.432,Z 777.951,A -85,B 0,C 180,E1 -454.638,E2 -454.638} C_VEL
LIN {X 0,Y 608.437,Z 771.877,A -85,B 0,C 180,E1 -455.801,E2 -455.801} C_VEL
LIN {X 0,Y 608.462,Z 765.236,A -85,B 0,C 180,E1 -456.799,E2 -456.799} C_VEL
LIN {X 0,Y 608.455,Z 756.991,A -85,B 0,C 180,E1 -457.8,E2 -457.8} C_VEL
LIN {X 0,Y 608.472,Z 748.539,A -85,B 0,C 180,E1 -458.636,E2 -458.636} C_VEL
LIN {X 0,Y 608.474,Z 738.094,A -85,B 0,C 180,E1 -459.473,E2 -459.473} C_VEL
LIN {X 0,Y 608.482,Z 727.76,A -85,B 0,C 180,E1 -460.145,E2 -460.145} C_VEL
LIN {X 0,Y 608.521,Z 716.245,A -85,B 0,C 180,E1 -460.741,E2 -460.741} C_VEL
LIN {X 0,Y 608.528,Z 704.883,A -85,B 0,C 180,E1 -461.192,E2 -461.192} C_VEL
LIN {X 0,Y 608.535,Z 692.28,A -85,B 0,C 180,E1 -461.554,E2 -461.554} C_VEL
LIN {X 0,Y 608.535,Z 679.622,A -85,B 0,C 180,E1 -461.787,E2 -461.787} C_VEL
LIN {X 0,Y 608.489,Z 574.948,A -85,B 0,C 180,E1 -463.037,E2 -463.037} C_VEL
LIN {X 0,Y 608.512,Z 550.733,A -85,B 0,C 180,E1 -465.92,E2 -465.92} C_VEL
LIN {X 0,Y 608.566,Z 526.338,A -85,B 0,C 180,E1 -468.866,E2 -468.866} C_VEL
LIN {X 0,Y 608.589,Z 503.378,A -85,B 0,C 180,E1 -471.687,E2 -471.687} C_VEL
LIN {X 0,Y 608.603,Z 484.346,A -85,B 0,C 180,E1 -474.067,E2 -474.067} C_VEL
LIN {X 0,Y 608.469,Z 483.687,A -85,B 0,C 180,E1 -474.197,E2 -474.197} C_VEL
LIN {X 0,Y 608.481,Z 483.695,A -85,B 0,C 180,E1 -477.207,E2 -477.207} C_VEL
LIN {X 0,Y 608.466,Z 483.686,A -85,B 0,C 180,E1 -479.971,E2 -479.971} C_VEL
LIN {X 0,Y 608.457,Z 483.688,A -85,B 0,C 180,E1 -482.521,E2 -482.521} C_VEL
LIN {X 0,Y 608.434,Z 483.699,A -85,B 0,C 180,E1 -485.277,E2 -485.277} C_VEL
LIN {X 0,Y 608.47,Z 483.687,A -85,B 0,C 180,E1 -487.745,E2 -487.745} C_VEL
LIN {X 0,Y 608.45,Z 483.688,A -85,B 0,C 180,E1 -490.329,E2 -490.329} C_VEL
LIN {X 0,Y 608.484,Z 483.692,A -85,B 0,C 180,E1 -493.31,E2 -493.31} C_VEL
LIN {X 0,Y 608.466,Z 483.685,A -85,B 0,C 180,E1 -496.13,E2 -496.13} C_VEL
LIN {X 0,Y 608.448,Z 483.692,A -85,B 0,C 180,E1 -498.823,E2 -498.823} C_VEL
LIN {X 0,Y 608.465,Z 483.692,A -85,B 0,C 180,E1 -501.412,E2 -501.412} C_VEL
LIN {X 0,Y 608.472,Z 483.685,A -85,B 0,C 180,E1 -503.949,E2 -503.949} C_VEL
LIN {X 0,Y 608.461,Z 483.686,A -85,B 0,C 180,E1 -506.329,E2 -506.329} C_VEL
LIN {X 0,Y 608.471,Z 483.688,A -85,B 0,C 180,E1 -508.726,E2 -508.726} C_VEL
LIN {X 0,Y 608.474,Z 483.691,A -85,B 0,C 180,E1 -511.377,E2 -511.377} C_VEL
LIN {X 0,Y 608.475,Z 483.684,A -85,B 0,C 180,E1 -514.276,E2 -514.276} C_VEL
LIN {X 0,Y 608.452,Z 483.693,A -85,B 0,C 180,E1 -516.876,E2 -516.876} C_VEL
LIN {X 0,Y 608.459,Z 483.688,A -85,B 0,C 180,E1 -519.726,E2 -519.726} C_VEL
LIN {X 0,Y 608.446,Z 483.689,A -85,B 0,C 180,E1 -522.523,E2 -522.523} C_VEL
LIN {X 0,Y 608.474,Z 483.692,A -85,B 0,C 180,E1 -525.28,E2 -525.28} C_VEL
LIN {X 0,Y 608.457,Z 483.687,A -85,B 0,C 180,E1 -528,E2 -528} C_VEL
LIN {X 0,Y 608.463,Z 483.689,A -85,B 0,C 180,E1 -530.694,E2 -530.694} C_VEL
LIN {X 0,Y 608.465,Z 483.692,A -85,B 0,C 180,E1 -533.367,E2 -533.367} C_VEL
LIN {X 0,Y 608.446,Z 483.688,A -85,B 0,C 180,E1 -536.026,E2 -536.026} C_VEL
LIN {X 0,Y 608.469,Z 483.689,A -85,B 0,C 180,E1 -538.676,E2 -538.676} C_VEL
LIN {X 0,Y 608.476,Z 483.691,A -85,B 0,C 180,E1 -541.324,E2 -541.324} C_VEL
LIN {X 0,Y 608.445,Z 483.688,A -85,B 0,C 180,E1 -543.974,E2 -543.974} C_VEL
LIN {X 0,Y 608.466,Z 483.689,A -85,B 0,C 180,E1 -546.633,E2 -546.633} C_VEL
LIN {X 0,Y 608.459,Z 483.69,A -85,B 0,C 180,E1 -549.472,E2 -549.472} C_VEL
LIN {X 0,Y 607.773,Z 483.774,A -85,B 0,C 180,E1 -550.025,E2 -550.025} C_VEL
LIN {X 0,Y 604.914,Z 484.136,A -85,B 0,C 180,E1 -550.922,E2 -550.922} C_VEL
LIN {X 0,Y 602.514,Z 484.43,A -85,B 0,C 180,E1 -551.643,E2 -551.643} C_VEL
LIN {X 0,Y 601.489,Z 484.555,A -85,B 0,C 180,E1 -552.2,E2 -552.2} C_VEL
LIN {X 0,Y 601.408,Z 484.566,A -85,B 0,C 180,E1 -552.388,E2 -552.388} C_VEL
LIN {X 0,Y 601.43,Z 484.569,A -85,B 0,C 180,E1 -554.897,E2 -554.897} C_VEL
LIN {X 0,Y 601.397,Z 484.567,A -85,B 0,C 180,E1 -557.689,E2 -557.689} C_VEL
LIN {X 0,Y 601.43,Z 484.564,A -85,B 0,C 180,E1 -560.522,E2 -560.522} C_VEL
LIN {X 0,Y 601.42,Z 484.567,A -85,B 0,C 180,E1 -563.411,E2 -563.411} C_VEL
LIN {X 0,Y 601.405,Z 484.566,A -85,B 0,C 180,E1 -566.364,E2 -566.364} C_VEL
LIN {X 0,Y 601.439,Z 484.567,A -85,B 0,C 180,E1 -568.792,E2 -568.792} C_VEL
LIN {X 0,Y 601.438,Z 484.565,A -85,B 0,C 180,E1 -571.46,E2 -571.46} C_VEL
LIN {X 0,Y 601.428,Z 484.562,A -85,B 0,C 180,E1 -574.119,E2 -574.119} C_VEL
LIN {X 0,Y 601.416,Z 484.567,A -85,B 0,C 180,E1 -576.583,E2 -576.583} C_VEL
LIN {X 0,Y 601.443,Z 484.563,A -85,B 0,C 180,E1 -579.538,E2 -579.538} C_VEL
LIN {X 0,Y 601.421,Z 484.564,A -85,B 0,C 180,E1 -581.766,E2 -581.766} C_VEL
LIN {X 0,Y 601.421,Z 484.566,A -85,B 0,C 180,E1 -584.536,E2 -584.536} C_VEL
LIN {X 0,Y 601.438,Z 484.565,A -85,B 0,C 180,E1 -587.407,E2 -587.407} C_VEL
LIN {X 0,Y 601.439,Z 484.563,A -85,B 0,C 180,E1 -590.465,E2 -590.465} C_VEL
LIN {X 0,Y 601.406,Z 484.569,A -85,B 0,C 180,E1 -593.418,E2 -593.418} C_VEL
LIN {X 0,Y 601.433,Z 484.562,A -85,B 0,C 180,E1 -596.065,E2 -596.065} C_VEL
LIN {X 0,Y 601.431,Z 484.565,A -85,B 0,C 180,E1 -598.545,E2 -598.545} C_VEL
LIN {X 0,Y 601.431,Z 484.566,A -85,B 0,C 180,E1 -601.374,E2 -601.374} C_VEL
LIN {X 0,Y 601.403,Z 484.567,A -85,B 0,C 180,E1 -603.637,E2 -603.637} C_VEL
LIN {X 0,Y 601.435,Z 484.622,A -85,B 0,C 180,E1 -606.043,E2 -606.043} C_VEL
LIN {X 0,Y 601.591,Z 494.235,A -85,B 0,C 180,E1 -607.459,E2 -607.459} C_VEL
LIN {X 0,Y 601.511,Z 513.149,A -85,B 0,C 180,E1 -610.195,E2 -610.195} C_VEL
LIN {X 0,Y 601.497,Z 532.946,A -85,B 0,C 180,E1 -613.016,E2 -613.016} C_VEL
LIN {X 0,Y 601.472,Z 546.365,A -85,B 0,C 180,E1 -614.877,E2 -614.877} C_VEL
LIN {X 0,Y 601.653,Z 596.021,A -85,B 0,C 180,E1 -615.477,E2 -615.477} C_VEL
LIN {X 0,Y 601.603,Z 654.799,A -85,B 0,C 180,E1 -616.2,E2 -616.2} C_VEL
LIN {X 0,Y 601.563,Z 668.179,A -85,B 0,C 180,E1 -616.509,E2 -616.509} C_VEL
LIN {X 0,Y 601.548,Z 681.22,A -85,B 0,C 180,E1 -616.96,E2 -616.96} C_VEL
LIN {X 0,Y 601.515,Z 693.05,A -85,B 0,C 180,E1 -617.517,E2 -617.517} C_VEL
LIN {X 0,Y 601.487,Z 704.414,A -85,B 0,C 180,E1 -618.201,E2 -618.201} C_VEL
LIN {X 0,Y 601.443,Z 714.807,A -85,B 0,C 180,E1 -618.982,E2 -618.982} C_VEL
LIN {X 0,Y 601.425,Z 724.658,A -85,B 0,C 180,E1 -619.905,E2 -619.905} C_VEL
LIN {X 0,Y 601.393,Z 733.445,A -85,B 0,C 180,E1 -620.923,E2 -620.923} C_VEL
LIN {X 0,Y 601.365,Z 740.454,A -85,B 0,C 180,E1 -621.938,E2 -621.938} C_VEL
LIN {X 0,Y 601.369,Z 746.055,A -85,B 0,C 180,E1 -622.952,E2 -622.952} C_VEL
LIN {X 0,Y 601.357,Z 750.451,A -85,B 0,C 180,E1 -623.962,E2 -623.962} C_VEL
LIN {X 0,Y 601.353,Z 752.768,A -85,B 0,C 180,E1 -624.635,E2 -624.635} C_VEL
LIN {X 0,Y 601.329,Z 754.658,A -85,B 0,C 180,E1 -625.307,E2 -625.307} C_VEL
LIN {X 0,Y 601.342,Z 756.108,A -85,B 0,C 180,E1 -625.979,E2 -625.979} C_VEL
LIN {X 0,Y 601.32,Z 757.745,A -85,B 0,C 180,E1 -627.32,E2 -627.32} C_VEL
LIN {X 0,Y 601.343,Z 757.994,A -85,B 0,C 180,E1 -627.991,E2 -627.991} C_VEL
LIN {X 0,Y 601.347,Z 757.821,A -85,B 0,C 180,E1 -628.661,E2 -628.661} C_VEL
LIN {X 0,Y 601.338,Z 756.29,A -85,B 0,C 180,E1 -630,E2 -630} C_VEL
LIN {X 0,Y 601.338,Z 754.94,A -85,B 0,C 180,E1 -630.67,E2 -630.67} C_VEL
LIN {X 0,Y 601.358,Z 752.076,A -85,B 0,C 180,E1 -631.674,E2 -631.674} C_VEL
LIN {X 0,Y 601.337,Z 748.198,A -85,B 0,C 180,E1 -632.679,E2 -632.679} C_VEL
LIN {X 0,Y 601.368,Z 743.196,A -85,B 0,C 180,E1 -633.685,E2 -633.685} C_VEL
LIN {X 0,Y 601.401,Z 736.921,A -85,B 0,C 180,E1 -634.692,E2 -634.692} C_VEL
LIN {X 0,Y 601.399,Z 729.078,A -85,B 0,C 180,E1 -635.701,E2 -635.701} C_VEL
LIN {X 0,Y 601.437,Z 719.32,A -85,B 0,C 180,E1 -636.71,E2 -636.71} C_VEL
LIN {X 0,Y 601.455,Z 709.14,A -85,B 0,C 180,E1 -637.554,E2 -637.554} C_VEL
LIN {X 0,Y 601.489,Z 697.688,A -85,B 0,C 180,E1 -638.314,E2 -638.314} C_VEL
LIN {X 0,Y 601.531,Z 686.386,A -85,B 0,C 180,E1 -638.905,E2 -638.905} C_VEL
LIN {X 0,Y 601.57,Z 674.821,A -85,B 0,C 180,E1 -639.371,E2 -639.371} C_VEL
LIN {X 0,Y 601.576,Z 661.541,A -85,B 0,C 180,E1 -639.753,E2 -639.753} C_VEL
LIN {X 0,Y 601.613,Z 648.492,A -85,B 0,C 180,E1 -639.986,E2 -639.986} C_VEL
LIN {X 0,Y 601.511,Z 546.566,A -85,B 0,C 180,E1 -641.21,E2 -641.21} C_VEL
LIN {X 0,Y 601.457,Z 545.729,A -85,B 0,C 180,E1 -641.272,E2 -641.272} C_VEL
LIN {X 0,Y 601.512,Z 524.987,A -85,B 0,C 180,E1 -644.203,E2 -644.203} C_VEL
LIN {X 0,Y 601.559,Z 505.597,A -85,B 0,C 180,E1 -646.982,E2 -646.982} C_VEL
LIN {X 0,Y 601.618,Z 487.451,A -85,B 0,C 180,E1 -649.624,E2 -649.624} C_VEL
LIN {X 0,Y 601.412,Z 484.568,A -85,B 0,C 180,E1 -650.076,E2 -650.076} C_VEL
LIN {X 0,Y 601.415,Z 484.569,A -85,B 0,C 180,E1 -652.682,E2 -652.682} C_VEL
LIN {X 0,Y 601.405,Z 484.573,A -85,B 0,C 180,E1 -654.878,E2 -654.878} C_VEL
LIN {X 0,Y 601.421,Z 484.568,A -85,B 0,C 180,E1 -657.362,E2 -657.362} C_VEL
LIN {X 0,Y 601.43,Z 484.563,A -85,B 0,C 180,E1 -660.163,E2 -660.163} C_VEL
LIN {X 0,Y 601.423,Z 484.569,A -85,B 0,C 180,E1 -662.715,E2 -662.715} C_VEL
LIN {X 0,Y 601.398,Z 484.574,A -85,B 0,C 180,E1 -665.111,E2 -665.111} C_VEL
LIN {X 0,Y 601.436,Z 484.564,A -85,B 0,C 180,E1 -667.418,E2 -667.418} C_VEL
LIN {X 0,Y 601.412,Z 484.564,A -85,B 0,C 180,E1 -669.994,E2 -669.994} C_VEL
LIN {X 0,Y 601.438,Z 484.568,A -85,B 0,C 180,E1 -672.667,E2 -672.667} C_VEL
LIN {X 0,Y 601.423,Z 484.564,A -85,B 0,C 180,E1 -675.481,E2 -675.481} C_VEL
LIN {X 0,Y 601.424,Z 484.567,A -85,B 0,C 180,E1 -678.405,E2 -678.405} C_VEL
LIN {X 0,Y 601.433,Z 484.571,A -85,B 0,C 180,E1 -680.875,E2 -680.875} C_VEL
LIN {X 0,Y 601.438,Z 484.561,A -85,B 0,C 180,E1 -683.733,E2 -683.733} C_VEL
LIN {X 0,Y 601.432,Z 484.563,A -85,B 0,C 180,E1 -686.062,E2 -686.062} C_VEL
LIN {X 0,Y 601.45,Z 484.653,A -85,B 0,C 180,E1 -688.177,E2 -688.177} C_VEL
LIN {X 0,Y 601.406,Z 498.348,A -85,B 0,C 180,E1 -690.889,E2 -690.889} C_VEL
LIN {X 0,Y 601.683,Z 501.571,A -85,B 0,C 180,E1 -690.944,E2 -690.944} C_VEL
LIN {X 0,Y 601.591,Z 604.704,A -85,B 0,C 180,E1 -692.198,E2 -692.198} C_VEL
LIN {X 0,Y 601.556,Z 618.806,A -85,B 0,C 180,E1 -692.527,E2 -692.527} C_VEL
LIN {X 0,Y 601.559,Z 630.735,A -85,B 0,C 180,E1 -692.941,E2 -692.941} C_VEL
LIN {X 0,Y 601.496,Z 641.849,A -85,B 0,C 180,E1 -693.453,E2 -693.453} C_VEL
LIN {X 0,Y 601.484,Z 653.12,A -85,B 0,C 180,E1 -694.116,E2 -694.116} C_VEL
LIN {X 0,Y 601.463,Z 664.28,A -85,B 0,C 180,E1 -694.939,E2 -694.939} C_VEL
LIN {X 0,Y 601.394,Z 674.191,A -85,B 0,C 180,E1 -695.857,E2 -695.857} C_VEL
LIN {X 0,Y 601.384,Z 682.222,A -85,B 0,C 180,E1 -696.77,E2 -696.77} C_VEL
LIN {X 0,Y 601.382,Z 689.064,A -85,B 0,C 180,E1 -697.721,E2 -697.721} C_VEL
LIN {X 0,Y 601.378,Z 695.097,A -85,B 0,C 180,E1 -698.759,E2 -698.759} C_VEL
LIN {X 0,Y 601.355,Z 699.967,A -85,B 0,C 180,E1 -699.832,E2 -699.832} C_VEL
LIN {X 0,Y 601.338,Z 703.577,A -85,B 0,C 180,E1 -700.898,E2 -700.898} C_VEL
LIN {X 0,Y 601.32,Z 705.336,A -85,B 0,C 180,E1 -701.605,E2 -701.605} C_VEL
LIN {X 0,Y 601.312,Z 706.649,A -85,B 0,C 180,E1 -702.309,E2 -702.309} C_VEL
LIN {X 0,Y 601.321,Z 707.804,A -85,B 0,C 180,E1 -703.407,E2 -703.407} C_VEL
LIN {X 0,Y 601.326,Z 707.919,A -85,B 0,C 180,E1 -704.406,E2 -704.406} C_VEL
LIN {X 0,Y 601.313,Z 707.507,A -85,B 0,C 180,E1 -705.1,E2 -705.1} C_VEL
LIN {X 0,Y 601.338,Z 706.4,A -85,B 0,C 180,E1 -705.935,E2 -705.935} C_VEL
LIN {X 0,Y 601.327,Z 703.638,A -85,B 0,C 180,E1 -707.17,E2 -707.17} C_VEL
LIN {X 0,Y 601.346,Z 700.192,A -85,B 0,C 180,E1 -708.198,E2 -708.198} C_VEL
LIN {X 0,Y 601.339,Z 695.651,A -85,B 0,C 180,E1 -709.222,E2 -709.222} C_VEL
LIN {X 0,Y 601.385,Z 688.778,A -85,B 0,C 180,E1 -710.414,E2 -710.414} C_VEL
LIN {X 0,Y 601.404,Z 681.331,A -85,B 0,C 180,E1 -711.431,E2 -711.431} C_VEL
LIN {X 0,Y 601.412,Z 672.088,A -85,B 0,C 180,E1 -712.446,E2 -712.446} C_VEL
LIN {X 0,Y 601.448,Z 662.152,A -85,B 0,C 180,E1 -713.32,E2 -713.32} C_VEL
LIN {X 0,Y 601.464,Z 652.018,A -85,B 0,C 180,E1 -714.047,E2 -714.047} C_VEL
LIN {X 0,Y 601.539,Z 640.19,A -85,B 0,C 180,E1 -714.721,E2 -714.721} C_VEL
LIN {X 0,Y 601.56,Z 627.648,A -85,B 0,C 180,E1 -715.267,E2 -715.267} C_VEL
LIN {X 0,Y 601.597,Z 615.836,A -85,B 0,C 180,E1 -715.645,E2 -715.645} C_VEL
LIN {X 0,Y 601.627,Z 603.214,A -85,B 0,C 180,E1 -715.918,E2 -715.918} C_VEL
LIN {X 0,Y 601.547,Z 499.41,A -85,B 0,C 180,E1 -717.175,E2 -717.175} C_VEL
LIN {X 0,Y 601.416,Z 498.376,A -85,B 0,C 180,E1 -717.195,E2 -717.195} C_VEL
LIN {X 0,Y 601.426,Z 484.565,A -85,B 0,C 180,E1 -719.958,E2 -719.958} C_VEL
LIN {X 0,Y 601.447,Z 484.562,A -85,B 0,C 180,E1 -722.679,E2 -722.679} C_VEL
LIN {X 0,Y 601.435,Z 484.572,A -85,B 0,C 180,E1 -725.364,E2 -725.364} C_VEL
LIN {X 0,Y 601.435,Z 484.562,A -85,B 0,C 180,E1 -728.061,E2 -728.061} C_VEL
LIN {X 0,Y 601.424,Z 484.569,A -85,B 0,C 180,E1 -731.018,E2 -731.018} C_VEL
LIN {X 0,Y 601.418,Z 484.57,A -85,B 0,C 180,E1 -733.516,E2 -733.516} C_VEL
LIN {X 0,Y 601.434,Z 484.562,A -85,B 0,C 180,E1 -736.287,E2 -736.287} C_VEL
LIN {X 0,Y 601.416,Z 484.573,A -85,B 0,C 180,E1 -739.099,E2 -739.099} C_VEL
LIN {X 0,Y 601.408,Z 484.575,A -85,B 0,C 180,E1 -741.239,E2 -741.239} C_VEL
LIN {X 0,Y 601.449,Z 484.56,A -85,B 0,C 180,E1 -744.141,E2 -744.141} C_VEL
LIN {X 0,Y 601.453,Z 484.57,A -85,B 0,C 180,E1 -747.111,E2 -747.111} C_VEL
LIN {X 0,Y 601.42,Z 484.569,A -85,B 0,C 180,E1 -749.393,E2 -749.393} C_VEL
LIN {X 0,Y 601.408,Z 484.566,A -85,B 0,C 180,E1 -751.727,E2 -751.727} C_VEL
LIN {X 0,Y 601.427,Z 484.562,A -85,B 0,C 180,E1 -754.119,E2 -754.119} C_VEL
LIN {X 0,Y 601.415,Z 484.567,A -85,B 0,C 180,E1 -756.582,E2 -756.582} C_VEL
LIN {X 0,Y 601.441,Z 484.563,A -85,B 0,C 180,E1 -759.537,E2 -759.537} C_VEL
LIN {X 0,Y 601.406,Z 484.569,A -85,B 0,C 180,E1 -762.592,E2 -762.592} C_VEL
LIN {X 0,Y 601.421,Z 484.566,A -85,B 0,C 180,E1 -765.483,E2 -765.483} C_VEL
LIN {X 0,Y 601.423,Z 484.566,A -85,B 0,C 180,E1 -768.407,E2 -768.407} C_VEL
LIN {X 0,Y 601.435,Z 484.572,A -85,B 0,C 180,E1 -770.876,E2 -770.876} C_VEL
LIN {X 0,Y 601.429,Z 484.563,A -85,B 0,C 180,E1 -773.736,E2 -773.736} C_VEL
LIN {X 0,Y 601.425,Z 484.57,A -85,B 0,C 180,E1 -776.687,E2 -776.687} C_VEL
LIN {X 0,Y 601.431,Z 484.569,A -85,B 0,C 180,E1 -779.06,E2 -779.06} C_VEL
LIN {X 0,Y 601.426,Z 484.565,A -85,B 0,C 180,E1 -781.374,E2 -781.374} C_VEL
LIN {X 0,Y 601.4,Z 484.567,A -85,B 0,C 180,E1 -783.637,E2 -783.637} C_VEL
LIN {X 0,Y 601.446,Z 484.571,A -85,B 0,C 180,E1 -785.657,E2 -785.657} C_VEL
LIN {X 0,Y 601.757,Z 487.593,A -85,B 0,C 180,E1 -786.056,E2 -786.056} C_VEL
LIN {X 0,Y 601.693,Z 509.118,A -85,B 0,C 180,E1 -788.772,E2 -788.772} C_VEL
LIN {X 0,Y 601.601,Z 533.513,A -85,B 0,C 180,E1 -791.791,E2 -791.791} C_VEL
LIN {X 0,Y 601.529,Z 556.473,A -85,B 0,C 180,E1 -794.586,E2 -794.586} C_VEL
LIN {X 0,Y 601.505,Z 575.275,A -85,B 0,C 180,E1 -796.82,E2 -796.82} C_VEL
LIN {X 0,Y 601.603,Z 683.962,A -85,B 0,C 180,E1 -798.14,E2 -798.14} C_VEL
LIN {X 0,Y 601.579,Z 697.225,A -85,B 0,C 180,E1 -798.438,E2 -798.438} C_VEL
LIN {X 0,Y 601.547,Z 708.925,A -85,B 0,C 180,E1 -798.826,E2 -798.826} C_VEL
LIN {X 0,Y 601.515,Z 719.929,A -85,B 0,C 180,E1 -799.311,E2 -799.311} C_VEL
LIN {X 0,Y 601.466,Z 730.584,A -85,B 0,C 180,E1 -799.906,E2 -799.906} C_VEL
LIN {X 0,Y 601.445,Z 741.478,A -85,B 0,C 180,E1 -800.67,E2 -800.67} C_VEL
LIN {X 0,Y 601.429,Z 752.114,A -85,B 0,C 180,E1 -801.601,E2 -801.601} C_VEL
LIN {X 0,Y 601.418,Z 759.962,A -85,B 0,C 180,E1 -802.446,E2 -802.446} C_VEL
LIN {X 0,Y 601.37,Z 767.225,A -85,B 0,C 180,E1 -803.398,E2 -803.398} C_VEL
LIN {X 0,Y 601.371,Z 772.867,A -85,B 0,C 180,E1 -804.299,E2 -804.299} C_VEL
LIN {X 0,Y 601.337,Z 777.95,A -85,B 0,C 180,E1 -805.307,E2 -805.307} C_VEL
LIN {X 0,Y 601.367,Z 781.896,A -85,B 0,C 180,E1 -806.315,E2 -806.315} C_VEL
LIN {X 0,Y 601.325,Z 784.809,A -85,B 0,C 180,E1 -807.321,E2 -807.321} C_VEL
LIN {X 0,Y 601.34,Z 786.202,A -85,B 0,C 180,E1 -807.991,E2 -807.991} C_VEL
LIN {X 0,Y 601.339,Z 787.784,A -85,B 0,C 180,E1 -809.33,E2 -809.33} C_VEL
LIN {X 0,Y 601.335,Z 788,A -85,B 0,C 180,E1 -810,E2 -810} C_VEL
LIN {X 0,Y 601.348,Z 787.184,A -85,B 0,C 180,E1 -811.339,E2 -811.339} C_VEL
LIN {X 0,Y 601.34,Z 786.202,A -85,B 0,C 180,E1 -812.009,E2 -812.009} C_VEL
LIN {X 0,Y 601.325,Z 784.809,A -85,B 0,C 180,E1 -812.679,E2 -812.679} C_VEL
LIN {X 0,Y 601.367,Z 781.896,A -85,B 0,C 180,E1 -813.685,E2 -813.685} C_VEL
LIN {X 0,Y 601.337,Z 777.951,A -85,B 0,C 180,E1 -814.693,E2 -814.693} C_VEL
LIN {X 0,Y 601.372,Z 771.878,A -85,B 0,C 180,E1 -815.869,E2 -815.869} C_VEL
LIN {X 0,Y 601.382,Z 765.237,A -85,B 0,C 180,E1 -816.88,E2 -816.88} C_VEL
LIN {X 0,Y 601.4,Z 756.991,A -85,B 0,C 180,E1 -817.892,E2 -817.892} C_VEL
LIN {X 0,Y 601.436,Z 748.539,A -85,B 0,C 180,E1 -818.737,E2 -818.737} C_VEL
LIN {X 0,Y 601.442,Z 738.095,A -85,B 0,C 180,E1 -819.585,E2 -819.585} C_VEL
LIN {X 0,Y 601.484,Z 727.761,A -85,B 0,C 180,E1 -820.264,E2 -820.264} C_VEL
LIN {X 0,Y 601.537,Z 716.901,A -85,B 0,C 180,E1 -820.836,E2 -820.836} C_VEL
LIN {X 0,Y 601.559,Z 704.383,A -85,B 0,C 180,E1 -821.34,E2 -821.34} C_VEL
LIN {X 0,Y 601.59,Z 691.366,A -85,B 0,C 180,E1 -821.711,E2 -821.711} C_VEL
LIN {X 0,Y 601.61,Z 678.106,A -85,B 0,C 180,E1 -821.946,E2 -821.946} C_VEL
LIN {X 0,Y 601.505,Z 575.275,A -85,B 0,C 180,E1 -823.18,E2 -823.18} C_VEL
LIN {X 0,Y 601.522,Z 553.603,A -85,B 0,C 180,E1 -825.762,E2 -825.762} C_VEL
LIN {X 0,Y 601.612,Z 530.075,A -85,B 0,C 180,E1 -828.632,E2 -828.632} C_VEL
LIN {X 0,Y 601.703,Z 507.683,A -85,B 0,C 180,E1 -831.407,E2 -831.407} C_VEL
LIN {X 0,Y 601.755,Z 486.158,A -85,B 0,C 180,E1 -834.127,E2 -834.127} C_VEL
LIN {X 0,Y 601.426,Z 484.567,A -85,B 0,C 180,E1 -834.363,E2 -834.363} C_VEL
LIN {X 0,Y 601.453,Z 484.569,A -85,B 0,C 180,E1 -837.11,E2 -837.11} C_VEL
LIN {X 0,Y 601.414,Z 484.572,A -85,B 0,C 180,E1 -839.393,E2 -839.393} C_VEL
LIN {X 0,Y 601.412,Z 484.567,A -85,B 0,C 180,E1 -841.725,E2 -841.725} C_VEL
LIN {X 0,Y 601.425,Z 484.563,A -85,B 0,C 180,E1 -844.118,E2 -844.118} C_VEL
LIN {X 0,Y 601.435,Z 484.567,A -85,B 0,C 180,E1 -847.382,E2 -847.382} C_VEL
LIN {X 0,Y 601.408,Z 484.565,A -85,B 0,C 180,E1 -849.994,E2 -849.994} C_VEL
LIN {X 0,Y 601.411,Z 484.567,A -85,B 0,C 180,E1 -852.669,E2 -852.669} C_VEL
LIN {X 0,Y 601.42,Z 484.569,A -85,B 0,C 180,E1 -855.481,E2 -855.481} C_VEL
LIN {X 0,Y 601.418,Z 484.564,A -85,B 0,C 180,E1 -858.406,E2 -858.406} C_VEL
LIN {X 0,Y 601.431,Z 484.567,A -85,B 0,C 180,E1 -860.875,E2 -860.875} C_VEL
LIN {X 0,Y 601.437,Z 484.563,A -85,B 0,C 180,E1 -863.733,E2 -863.733} C_VEL
LIN {X 0,Y 601.429,Z 484.562,A -85,B 0,C 180,E1 -866.063,E2 -866.063} C_VEL
LIN {X 0,Y 601.435,Z 484.563,A -85,B 0,C 180,E1 -868.541,E2 -868.541} C_VEL
LIN {X 0,Y 601.433,Z 484.568,A -85,B 0,C 180,E1 -871.373,E2 -871.373} C_VEL
LIN {X 0,Y 601.416,Z 484.563,A -85,B 0,C 180,E1 -874.129,E2 -874.129} C_VEL
LIN {X 0,Y 601.418,Z 484.565,A -85,B 0,C 180,E1 -876.59,E2 -876.59} C_VEL
LIN {X 0,Y 601.43,Z 484.567,A -85,B 0,C 180,E1 -879.478,E2 -879.478} C_VEL
LIN {X 0,Y 601.392,Z 484.567,A -85,B 0,C 180,E1 -882.312,E2 -882.312} C_VEL
LIN {X 0,Y 601.408,Z 484.565,A -85,B 0,C 180,E1 -884.409,E2 -884.409} C_VEL
LIN {X 0,Y 601.421,Z 484.573,A -85,B 0,C 180,E1 -887.172,E2 -887.172} C_VEL
LIN {X 0,Y 601.429,Z 484.562,A -85,B 0,C 180,E1 -889.905,E2 -889.905} C_VEL
LIN {X 0,Y 601.444,Z 484.562,A -85,B 0,C 180,E1 -892.615,E2 -892.615} C_VEL
LIN {X 0,Y 601.432,Z 484.569,A -85,B 0,C 180,E1 -895.308,E2 -895.308} C_VEL
LIN {X 0,Y 601.416,Z 484.563,A -85,B 0,C 180,E1 -897.991,E2 -897.991} C_VEL
LIN {X 0,Y 601.451,Z 484.562,A -85,B 0,C 180,E1 -900.67,E2 -900.67} C_VEL
LIN {X 0,Y 601.436,Z 484.567,A -85,B 0,C 180,E1 -903.35,E2 -903.35} C_VEL
LIN {X 0,Y 601.426,Z 484.562,A -85,B 0,C 180,E1 -906.037,E2 -906.037} C_VEL
LIN {X 0,Y 601.437,Z 484.565,A -85,B 0,C 180,E1 -908.738,E2 -908.738} C_VEL
LIN {X 0,Y 601.432,Z 484.566,A -85,B 0,C 180,E1 -911.458,E2 -911.458} C_VEL
LIN {X 0,Y 601.408,Z 484.566,A -85,B 0,C 180,E1 -912.388,E2 -912.388} C_VEL
LIN {X 0,Y 600.747,Z 484.656,A -85,B 0,C 180,E1 -912.948,E2 -912.948} C_VEL
LIN {X 0,Y 597.898,Z 485.014,A -85,B 0,C 180,E1 -913.855,E2 -913.855} C_VEL
LIN {X 0,Y 595.485,Z 485.315,A -85,B 0,C 180,E1 -914.586,E2 -914.586} C_VEL
LIN {X 0,Y 594.446,Z 485.44,A -85,B 0,C 180,E1 -915.149,E2 -915.149} C_VEL
LIN {X 0,Y 594.361,Z 485.447,A -85,B 0,C 180,E1 -915.34,E2 -915.34} C_VEL
LIN {X 0,Y 594.377,Z 485.44,A -85,B 0,C 180,E1 -917.905,E2 -917.905} C_VEL
LIN {X 0,Y 594.38,Z 485.449,A -85,B 0,C 180,E1 -920.92,E2 -920.92} C_VEL
LIN {X 0,Y 594.387,Z 485.44,A -85,B 0,C 180,E1 -923.704,E2 -923.704} C_VEL
LIN {X 0,Y 594.387,Z 485.444,A -85,B 0,C 180,E1 -926.7,E2 -926.7} C_VEL
LIN {X 0,Y 594.381,Z 485.45,A -85,B 0,C 180,E1 -928.999,E2 -928.999} C_VEL
LIN {X 0,Y 594.388,Z 485.441,A -85,B 0,C 180,E1 -931.646,E2 -931.646} C_VEL
LIN {X 0,Y 594.397,Z 485.441,A -85,B 0,C 180,E1 -934.579,E2 -934.579} C_VEL
LIN {X 0,Y 594.385,Z 485.45,A -85,B 0,C 180,E1 -937.087,E2 -937.087} C_VEL
LIN {X 0,Y 594.376,Z 485.441,A -85,B 0,C 180,E1 -939.776,E2 -939.776} C_VEL
LIN {X 0,Y 594.365,Z 485.444,A -85,B 0,C 180,E1 -942.376,E2 -942.376} C_VEL
LIN {X 0,Y 594.361,Z 485.45,A -85,B 0,C 180,E1 -945.192,E2 -945.192} C_VEL
LIN {X 0,Y 594.386,Z 485.441,A -85,B 0,C 180,E1 -947.627,E2 -947.627} C_VEL
LIN {X 0,Y 594.391,Z 485.44,A -85,B 0,C 180,E1 -950.322,E2 -950.322} C_VEL
LIN {X 0,Y 594.385,Z 485.449,A -85,B 0,C 180,E1 -952.914,E2 -952.914} C_VEL
LIN {X 0,Y 594.383,Z 485.44,A -85,B 0,C 180,E1 -955.862,E2 -955.862} C_VEL
LIN {X 0,Y 594.382,Z 485.445,A -85,B 0,C 180,E1 -958.651,E2 -958.651} C_VEL
LIN {X 0,Y 594.384,Z 485.45,A -85,B 0,C 180,E1 -961.043,E2 -961.043} C_VEL
LIN {X 0,Y 594.388,Z 485.445,A -85,B 0,C 180,E1 -963.301,E2 -963.301} C_VEL
LIN {X 0,Y 594.425,Z 485.53,A -85,B 0,C 180,E1 -965.905,E2 -965.905} C_VEL
LIN {X 0,Y 594.671,Z 493.138,A -85,B 0,C 180,E1 -967.046,E2 -967.046} C_VEL
LIN {X 0,Y 594.563,Z 511.734,A -85,B 0,C 180,E1 -969.773,E2 -969.773} C_VEL
LIN {X 0,Y 594.49,Z 530.299,A -85,B 0,C 180,E1 -972.455,E2 -972.455} C_VEL
LIN {X 0,Y 594.414,Z 546.137,A -85,B 0,C 180,E1 -974.715,E2 -974.715} C_VEL
LIN {X 0,Y 594.758,Z 550.747,A -85,B 0,C 180,E1 -974.779,E2 -974.779} C_VEL
LIN {X 0,Y 594.653,Z 654.042,A -85,B 0,C 180,E1 -976.046,E2 -976.046} C_VEL
LIN {X 0,Y 594.641,Z 667.346,A -85,B 0,C 180,E1 -976.349,E2 -976.349} C_VEL
LIN {X 0,Y 594.585,Z 679.53,A -85,B 0,C 180,E1 -976.761,E2 -976.761} C_VEL
LIN {X 0,Y 594.538,Z 690.981,A -85,B 0,C 180,E1 -977.282,E2 -977.282} C_VEL
LIN {X 0,Y 594.463,Z 702.775,A -85,B 0,C 180,E1 -977.973,E2 -977.973} C_VEL
LIN {X 0,Y 594.414,Z 713.569,A -85,B 0,C 180,E1 -978.772,E2 -978.772} C_VEL
LIN {X 0,Y 594.38,Z 722.785,A -85,B 0,C 180,E1 -979.612,E2 -979.612} C_VEL
LIN {X 0,Y 594.315,Z 731.906,A -85,B 0,C 180,E1 -980.642,E2 -980.642} C_VEL
LIN {X 0,Y 594.288,Z 739.242,A -85,B 0,C 180,E1 -981.671,E2 -981.671} C_VEL
LIN {X 0,Y 594.292,Z 745.945,A -85,B 0,C 180,E1 -982.867,E2 -982.867} C_VEL
LIN {X 0,Y 594.26,Z 750.366,A -85,B 0,C 180,E1 -983.89,E2 -983.89} C_VEL
LIN {X 0,Y 594.271,Z 752.696,A -85,B 0,C 180,E1 -984.571,E2 -984.571} C_VEL
LIN {X 0,Y 594.229,Z 754.596,A -85,B 0,C 180,E1 -985.251,E2 -985.251} C_VEL
LIN {X 0,Y 594.255,Z 756.068,A -85,B 0,C 180,E1 -985.931,E2 -985.931} C_VEL
LIN {X 0,Y 594.259,Z 757.092,A -85,B 0,C 180,E1 -986.61,E2 -986.61} C_VEL
LIN {X 0,Y 594.242,Z 757.988,A -85,B 0,C 180,E1 -987.967,E2 -987.967} C_VEL
LIN {X 0,Y 594.247,Z 757.837,A -85,B 0,C 180,E1 -988.645,E2 -988.645} C_VEL
LIN {X 0,Y 594.238,Z 756.328,A -85,B 0,C 180,E1 -990,E2 -990} C_VEL
LIN {X 0,Y 594.239,Z 754.991,A -85,B 0,C 180,E1 -990.678,E2 -990.678} C_VEL
LIN {X 0,Y 594.28,Z 752.15,A -85,B 0,C 180,E1 -991.694,E2 -991.694} C_VEL
LIN {X 0,Y 594.243,Z 748.297,A -85,B 0,C 180,E1 -992.711,E2 -992.711} C_VEL
LIN {X 0,Y 594.289,Z 743.323,A -85,B 0,C 180,E1 -993.729,E2 -993.729} C_VEL
LIN {X 0,Y 594.339,Z 737.08,A -85,B 0,C 180,E1 -994.748,E2 -994.748} C_VEL
LIN {X 0,Y 594.33,Z 729.285,A -85,B 0,C 180,E1 -995.769,E2 -995.769} C_VEL
LIN {X 0,Y 594.393,Z 719.567,A -85,B 0,C 180,E1 -996.79,E2 -996.79} C_VEL
LIN {X 0,Y 594.433,Z 709.462,A -85,B 0,C 180,E1 -997.643,E2 -997.643} C_VEL
LIN {X 0,Y 594.497,Z 698.079,A -85,B 0,C 180,E1 -998.412,E2 -998.412} C_VEL
LIN {X 0,Y 594.545,Z 686.888,A -85,B 0,C 180,E1 -999.011,E2 -999.011} C_VEL
LIN {X 0,Y 594.622,Z 674.25,A -85,B 0,C 180,E1 -999.524,E2 -999.524} C_VEL
LIN {X 0,Y 594.607,Z 660.738,A -85,B 0,C 180,E1 -999.911,E2 -999.911} C_VEL
LIN {X 0,Y 594.653,Z 646.963,A -85,B 0,C 180,E1 -1000.147,E2 -1000.147} C_VEL
LIN {X 0,Y 594.679,Z 547.707,A -85,B 0,C 180,E1 -1001.35,E2 -1001.35} C_VEL
LIN {X 0,Y 594.429,Z 546.033,A -85,B 0,C 180,E1 -1001.388,E2 -1001.388} C_VEL
LIN {X 0,Y 594.497,Z 526.283,A -85,B 0,C 180,E1 -1004.212,E2 -1004.212} C_VEL
LIN {X 0,Y 594.581,Z 507.622,A -85,B 0,C 180,E1 -1006.916,E2 -1006.916} C_VEL
LIN {X 0,Y 594.685,Z 490.043,A -85,B 0,C 180,E1 -1009.503,E2 -1009.503} C_VEL
LIN {X 0,Y 594.392,Z 485.444,A -85,B 0,C 180,E1 -1010.21,E2 -1010.21} C_VEL
LIN {X 0,Y 594.359,Z 485.453,A -85,B 0,C 180,E1 -1012.967,E2 -1012.967} C_VEL
LIN {X 0,Y 594.376,Z 485.45,A -85,B 0,C 180,E1 -1015.192,E2 -1015.192} C_VEL
LIN {X 0,Y 594.388,Z 485.442,A -85,B 0,C 180,E1 -1017.526,E2 -1017.526} C_VEL
LIN {X 0,Y 594.39,Z 485.441,A -85,B 0,C 180,E1 -1020.328,E2 -1020.328} C_VEL
LIN {X 0,Y 594.378,Z 485.451,A -85,B 0,C 180,E1 -1022.949,E2 -1022.949} C_VEL
LIN {X 0,Y 594.351,Z 485.447,A -85,B 0,C 180,E1 -1025.408,E2 -1025.408} C_VEL
LIN {X 0,Y 594.389,Z 485.439,A -85,B 0,C 180,E1 -1027.939,E2 -1027.939} C_VEL
LIN {X 0,Y 594.382,Z 485.449,A -85,B 0,C 180,E1 -1030.822,E2 -1030.822} C_VEL
LIN {X 0,Y 594.385,Z 485.443,A -85,B 0,C 180,E1 -1033.297,E2 -1033.297} C_VEL
LIN {X 0,Y 594.379,Z 485.441,A -85,B 0,C 180,E1 -1036.158,E2 -1036.158} C_VEL
LIN {X 0,Y 594.377,Z 485.445,A -85,B 0,C 180,E1 -1039.176,E2 -1039.176} C_VEL
LIN {X 0,Y 594.382,Z 485.441,A -85,B 0,C 180,E1 -1042.058,E2 -1042.058} C_VEL
LIN {X 0,Y 594.383,Z 485.449,A -85,B 0,C 180,E1 -1044.67,E2 -1044.67} C_VEL
LIN {X 0,Y 594.374,Z 485.447,A -85,B 0,C 180,E1 -1047.087,E2 -1047.087} C_VEL
LIN {X 0,Y 594.413,Z 485.572,A -85,B 0,C 180,E1 -1048.17,E2 -1048.17} C_VEL
LIN {X 0,Y 594.374,Z 498.577,A -85,B 0,C 180,E1 -1050.744,E2 -1050.744} C_VEL
LIN {X 0,Y 594.771,Z 502.815,A -85,B 0,C 180,E1 -1050.804,E2 -1050.804} C_VEL
LIN {X 0,Y 594.664,Z 603.604,A -85,B 0,C 180,E1 -1052.04,E2 -1052.04} C_VEL
LIN {X 0,Y 594.611,Z 616.779,A -85,B 0,C 180,E1 -1052.333,E2 -1052.333} C_VEL
LIN {X 0,Y 594.554,Z 630.183,A -85,B 0,C 180,E1 -1052.786,E2 -1052.786} C_VEL
LIN {X 0,Y 594.524,Z 641.448,A -85,B 0,C 180,E1 -1053.307,E2 -1053.307} C_VEL
LIN {X 0,Y 594.457,Z 652.572,A -85,B 0,C 180,E1 -1053.961,E2 -1053.961} C_VEL
LIN {X 0,Y 594.421,Z 662.857,A -85,B 0,C 180,E1 -1054.715,E2 -1054.715} C_VEL
LIN {X 0,Y 594.387,Z 672.301,A -85,B 0,C 180,E1 -1055.564,E2 -1055.564} C_VEL
LIN {X 0,Y 594.331,Z 680.586,A -85,B 0,C 180,E1 -1056.478,E2 -1056.478} C_VEL
LIN {X 0,Y 594.296,Z 688.232,A -85,B 0,C 180,E1 -1057.519,E2 -1057.519} C_VEL
LIN {X 0,Y 594.291,Z 694.012,A -85,B 0,C 180,E1 -1058.494,E2 -1058.494} C_VEL
LIN {X 0,Y 594.278,Z 699.135,A -85,B 0,C 180,E1 -1059.581,E2 -1059.581} C_VEL
LIN {X 0,Y 594.259,Z 702.975,A -85,B 0,C 180,E1 -1060.662,E2 -1060.662} C_VEL
LIN {X 0,Y 594.249,Z 704.898,A -85,B 0,C 180,E1 -1061.378,E2 -1061.378} C_VEL
LIN {X 0,Y 594.207,Z 706.327,A -85,B 0,C 180,E1 -1062.09,E2 -1062.09} C_VEL
LIN {X 0,Y 594.235,Z 707.752,A -85,B 0,C 180,E1 -1063.328,E2 -1063.328} C_VEL
LIN {X 0,Y 594.251,Z 707.961,A -85,B 0,C 180,E1 -1064.216,E2 -1064.216} C_VEL
LIN {X 0,Y 594.225,Z 707.654,A -85,B 0,C 180,E1 -1064.918,E2 -1064.918} C_VEL
LIN {X 0,Y 594.249,Z 706.536,A -85,B 0,C 180,E1 -1065.875,E2 -1065.875} C_VEL
LIN {X 0,Y 594.243,Z 704.144,A -85,B 0,C 180,E1 -1067.014,E2 -1067.014} C_VEL
LIN {X 0,Y 594.259,Z 700.894,A -85,B 0,C 180,E1 -1068.055,E2 -1068.055} C_VEL
LIN {X 0,Y 594.243,Z 696.565,A -85,B 0,C 180,E1 -1069.092,E2 -1069.092} C_VEL
LIN {X 0,Y 594.28,Z 691.035,A -85,B 0,C 180,E1 -1070.126,E2 -1070.126} C_VEL
LIN {X 0,Y 594.339,Z 684.132,A -85,B 0,C 180,E1 -1071.157,E2 -1071.157} C_VEL
LIN {X 0,Y 594.342,Z 675.597,A -85,B 0,C 180,E1 -1072.184,E2 -1072.184} C_VEL
LIN {X 0,Y 594.399,Z 666.826,A -85,B 0,C 180,E1 -1073.039,E2 -1073.039} C_VEL
LIN {X 0,Y 594.474,Z 656.058,A -85,B 0,C 180,E1 -1073.892,E2 -1073.892} C_VEL
LIN {X 0,Y 594.503,Z 645.305,A -85,B 0,C 180,E1 -1074.573,E2 -1074.573} C_VEL
LIN {X 0,Y 594.553,Z 633.363,A -85,B 0,C 180,E1 -1075.169,E2 -1075.169} C_VEL
LIN {X 0,Y 594.61,Z 620.906,A -85,B 0,C 180,E1 -1075.636,E2 -1075.636} C_VEL
LIN {X 0,Y 594.659,Z 607.692,A -85,B 0,C 180,E1 -1075.976,E2 -1075.976} C_VEL
LIN {X 0,Y 594.686,Z 589.965,A -85,B 0,C 180,E1 -1076.231,E2 -1076.231} C_VEL
LIN {X 0,Y 594.628,Z 500.098,A -85,B 0,C 180,E1 -1077.322,E2 -1077.322} C_VEL
LIN {X 0,Y 594.344,Z 498.28,A -85,B 0,C 180,E1 -1077.374,E2 -1077.374} C_VEL
LIN {X 0,Y 594.395,Z 485.442,A -85,B 0,C 180,E1 -1079.958,E2 -1079.958} C_VEL
LIN {X 0,Y 594.411,Z 485.439,A -85,B 0,C 180,E1 -1082.711,E2 -1082.711} C_VEL
LIN {X 0,Y 594.399,Z 485.447,A -85,B 0,C 180,E1 -1085.428,E2 -1085.428} C_VEL
LIN {X 0,Y 594.411,Z 485.437,A -85,B 0,C 180,E1 -1088.157,E2 -1088.157} C_VEL
LIN {X 0,Y 594.387,Z 485.447,A -85,B 0,C 180,E1 -1091.079,E2 -1091.079} C_VEL
LIN {X 0,Y 594.379,Z 485.444,A -85,B 0,C 180,E1 -1093.679,E2 -1093.679} C_VEL
LIN {X 0,Y 594.389,Z 485.442,A -85,B 0,C 180,E1 -1096.722,E2 -1096.722} C_VEL
LIN {X 0,Y 594.365,Z 485.451,A -85,B 0,C 180,E1 -1099.334,E2 -1099.334} C_VEL
LIN {X 0,Y 594.365,Z 485.447,A -85,B 0,C 180,E1 -1101.503,E2 -1101.503} C_VEL
LIN {X 0,Y 594.379,Z 485.441,A -85,B 0,C 180,E1 -1104.446,E2 -1104.446} C_VEL
LIN {X 0,Y 594.386,Z 485.443,A -85,B 0,C 180,E1 -1106.699,E2 -1106.699} C_VEL
LIN {X 0,Y 594.38,Z 485.449,A -85,B 0,C 180,E1 -1108.999,E2 -1108.999} C_VEL
LIN {X 0,Y 594.386,Z 485.441,A -85,B 0,C 180,E1 -1111.646,E2 -1111.646} C_VEL
LIN {X 0,Y 594.396,Z 485.441,A -85,B 0,C 180,E1 -1114.579,E2 -1114.579} C_VEL
LIN {X 0,Y 594.383,Z 485.45,A -85,B 0,C 180,E1 -1117.087,E2 -1117.087} C_VEL
LIN {X 0,Y 594.374,Z 485.442,A -85,B 0,C 180,E1 -1119.776,E2 -1119.776} C_VEL
LIN {X 0,Y 594.363,Z 485.444,A -85,B 0,C 180,E1 -1122.376,E2 -1122.376} C_VEL
LIN {X 0,Y 594.359,Z 485.45,A -85,B 0,C 180,E1 -1125.192,E2 -1125.192} C_VEL
LIN {X 0,Y 594.369,Z 485.443,A -85,B 0,C 180,E1 -1127.626,E2 -1127.626} C_VEL
LIN {X 0,Y 594.389,Z 485.441,A -85,B 0,C 180,E1 -1130.322,E2 -1130.322} C_VEL
LIN {X 0,Y 594.383,Z 485.451,A -85,B 0,C 180,E1 -1132.914,E2 -1132.914} C_VEL
LIN {X 0,Y 594.379,Z 485.441,A -85,B 0,C 180,E1 -1135.862,E2 -1135.862} C_VEL
LIN {X 0,Y 594.39,Z 485.447,A -85,B 0,C 180,E1 -1138.652,E2 -1138.652} C_VEL
LIN {X 0,Y 594.381,Z 485.448,A -85,B 0,C 180,E1 -1141.043,E2 -1141.043} C_VEL
LIN {X 0,Y 594.381,Z 485.442,A -85,B 0,C 180,E1 -1143.979,E2 -1143.979} C_VEL
LIN {X 0,Y 594.383,Z 485.514,A -85,B 0,C 180,E1 -1145.471,E2 -1145.471} C_VEL
LIN {X 0,Y 594.897,Z 489.028,A -85,B 0,C 180,E1 -1145.948,E2 -1145.948} C_VEL
LIN {X 0,Y 594.785,Z 510.407,A -85,B 0,C 180,E1 -1148.676,E2 -1148.676} C_VEL
LIN {X 0,Y 594.646,Z 532.078,A -85,B 0,C 180,E1 -1151.392,E2 -1151.392} C_VEL
LIN {X 0,Y 594.55,Z 555.038,A -85,B 0,C 180,E1 -1154.224,E2 -1154.224} C_VEL
LIN {X 0,Y 594.479,Z 575.275,A -85,B 0,C 180,E1 -1156.661,E2 -1156.661} C_VEL
LIN {X 0,Y 594.749,Z 581.535,A -85,B 0,C 180,E1 -1156.743,E2 -1156.743} C_VEL
LIN {X 0,Y 594.654,Z 683.962,A -85,B 0,C 180,E1 -1157.999,E2 -1157.999} C_VEL
LIN {X 0,Y 594.621,Z 697.225,A -85,B 0,C 180,E1 -1158.301,E2 -1158.301} C_VEL
LIN {X 0,Y 594.591,Z 710.375,A -85,B 0,C 180,E1 -1158.75,E2 -1158.75} C_VEL
LIN {X 0,Y 594.538,Z 721.638,A -85,B 0,C 180,E1 -1159.27,E2 -1159.27} C_VEL
LIN {X 0,Y 594.468,Z 733.203,A -85,B 0,C 180,E1 -1159.958,E2 -1159.958} C_VEL
LIN {X 0,Y 594.413,Z 743.598,A -85,B 0,C 180,E1 -1160.73,E2 -1160.73} C_VEL
LIN {X 0,Y 594.383,Z 752.114,A -85,B 0,C 180,E1 -1161.501,E2 -1161.501} C_VEL
LIN {X 0,Y 594.347,Z 759.962,A -85,B 0,C 180,E1 -1162.356,E2 -1162.356} C_VEL
LIN {X 0,Y 594.282,Z 767.813,A -85,B 0,C 180,E1 -1163.408,E2 -1163.408} C_VEL
LIN {X 0,Y 594.289,Z 774.681,A -85,B 0,C 180,E1 -1164.571,E2 -1164.571} C_VEL
LIN {X 0,Y 594.27,Z 779.371,A -85,B 0,C 180,E1 -1165.591,E2 -1165.591} C_VEL
LIN {X 0,Y 594.268,Z 782.957,A -85,B 0,C 180,E1 -1166.61,E2 -1166.61} C_VEL
LIN {X 0,Y 594.226,Z 784.81,A -85,B 0,C 180,E1 -1167.288,E2 -1167.288} C_VEL
LIN {X 0,Y 594.239,Z 786.202,A -85,B 0,C 180,E1 -1167.967,E2 -1167.967} C_VEL
LIN {X 0,Y 594.239,Z 787.784,A -85,B 0,C 180,E1 -1169.322,E2 -1169.322} C_VEL
LIN {X 0,Y 594.236,Z 788,A -85,B 0,C 180,E1 -1170,E2 -1170} C_VEL
LIN {X 0,Y 594.247,Z 787.184,A -85,B 0,C 180,E1 -1171.355,E2 -1171.355} C_VEL
LIN {X 0,Y 594.239,Z 786.202,A -85,B 0,C 180,E1 -1172.033,E2 -1172.033} C_VEL
LIN {X 0,Y 594.226,Z 784.809,A -85,B 0,C 180,E1 -1172.712,E2 -1172.712} C_VEL
LIN {X 0,Y 594.288,Z 781.896,A -85,B 0,C 180,E1 -1173.729,E2 -1173.729} C_VEL
LIN {X 0,Y 594.242,Z 777.95,A -85,B 0,C 180,E1 -1174.749,E2 -1174.749} C_VEL
LIN {X 0,Y 594.304,Z 771.878,A -85,B 0,C 180,E1 -1175.939,E2 -1175.939} C_VEL
LIN {X 0,Y 594.308,Z 765.237,A -85,B 0,C 180,E1 -1176.962,E2 -1176.962} C_VEL
LIN {X 0,Y 594.359,Z 756.991,A -85,B 0,C 180,E1 -1177.986,E2 -1177.986} C_VEL
LIN {X 0,Y 594.382,Z 748.539,A -85,B 0,C 180,E1 -1178.842,E2 -1178.842} C_VEL
LIN {X 0,Y 594.423,Z 738.097,A -85,B 0,C 180,E1 -1179.699,E2 -1179.699} C_VEL
LIN {X 0,Y 594.485,Z 727.762,A -85,B 0,C 180,E1 -1180.386,E2 -1180.386} C_VEL
LIN {X 0,Y 594.56,Z 716.696,A -85,B 0,C 180,E1 -1180.974,E2 -1180.974} C_VEL
LIN {X 0,Y 594.594,Z 704.711,A -85,B 0,C 180,E1 -1181.464,E2 -1181.464} C_VEL
LIN {X 0,Y 594.635,Z 691.366,A -85,B 0,C 180,E1 -1181.85,E2 -1181.85} C_VEL
LIN {X 0,Y 594.689,Z 678.106,A -85,B 0,C 180,E1 -1182.087,E2 -1182.087} C_VEL
LIN {X 0,Y 594.613,Z 576.169,A -85,B 0,C 180,E1 -1183.325,E2 -1183.325} C_VEL
LIN {X 0,Y 594.477,Z 574.769,A -85,B 0,C 180,E1 -1183.372,E2 -1183.372} C_VEL
LIN {X 0,Y 594.569,Z 550.733,A -85,B 0,C 180,E1 -1186.304,E2 -1186.304} C_VEL
LIN {X 0,Y 594.678,Z 528.065,A -85,B 0,C 180,E1 -1189.108,E2 -1189.108} C_VEL
LIN {X 0,Y 594.83,Z 504.813,A -85,B 0,C 180,E1 -1192.032,E2 -1192.032} C_VEL
LIN {X 0,Y 594.837,Z 487.593,A -85,B 0,C 180,E1 -1194.24,E2 -1194.24} C_VEL
LIN {X 0,Y 594.371,Z 485.449,A -85,B 0,C 180,E1 -1194.572,E2 -1194.572} C_VEL
LIN {X 0,Y 594.374,Z 485.448,A -85,B 0,C 180,E1 -1197.46,E2 -1197.46} C_VEL
LIN {X 0,Y 594.387,Z 485.44,A -85,B 0,C 180,E1 -1200.328,E2 -1200.328} C_VEL
LIN {X 0,Y 594.377,Z 485.447,A -85,B 0,C 180,E1 -1202.949,E2 -1202.949} C_VEL
LIN {X 0,Y 594.346,Z 485.451,A -85,B 0,C 180,E1 -1205.408,E2 -1205.408} C_VEL
LIN {X 0,Y 594.386,Z 485.438,A -85,B 0,C 180,E1 -1207.94,E2 -1207.94} C_VEL
LIN {X 0,Y 594.376,Z 485.445,A -85,B 0,C 180,E1 -1210.822,E2 -1210.822} C_VEL
LIN {X 0,Y 594.378,Z 485.441,A -85,B 0,C 180,E1 -1213.84,E2 -1213.84} C_VEL
LIN {X 0,Y 594.361,Z 485.446,A -85,B 0,C 180,E1 -1216.7,E2 -1216.7} C_VEL
LIN {X 0,Y 594.365,Z 485.448,A -85,B 0,C 180,E1 -1219.433,E2 -1219.433} C_VEL
LIN {X 0,Y 594.382,Z 485.44,A -85,B 0,C 180,E1 -1222.391,E2 -1222.391} C_VEL
LIN {X 0,Y 594.383,Z 485.442,A -85,B 0,C 180,E1 -1224.67,E2 -1224.67} C_VEL
LIN {X 0,Y 594.372,Z 485.451,A -85,B 0,C 180,E1 -1227.087,E2 -1227.087} C_VEL
LIN {X 0,Y 594.393,Z 485.441,A -85,B 0,C 180,E1 -1229.669,E2 -1229.669} C_VEL
LIN {X 0,Y 594.364,Z 485.444,A -85,B 0,C 180,E1 -1232.539,E2 -1232.539} C_VEL
LIN {X 0,Y 594.374,Z 485.445,A -85,B 0,C 180,E1 -1234.807,E2 -1234.807} C_VEL
LIN {X 0,Y 594.358,Z 485.451,A -85,B 0,C 180,E1 -1237.263,E2 -1237.263} C_VEL
LIN {X 0,Y 594.371,Z 485.442,A -85,B 0,C 180,E1 -1239.946,E2 -1239.946} C_VEL
LIN {X 0,Y 594.384,Z 485.444,A -85,B 0,C 180,E1 -1242.807,E2 -1242.807} C_VEL
LIN {X 0,Y 594.378,Z 485.441,A -85,B 0,C 180,E1 -1245.826,E2 -1245.826} C_VEL
LIN {X 0,Y 594.385,Z 485.44,A -85,B 0,C 180,E1 -1248.404,E2 -1248.404} C_VEL
LIN {X 0,Y 594.396,Z 485.447,A -85,B 0,C 180,E1 -1251.158,E2 -1251.158} C_VEL
LIN {X 0,Y 594.38,Z 485.44,A -85,B 0,C 180,E1 -1253.891,E2 -1253.891} C_VEL
LIN {X 0,Y 594.377,Z 485.443,A -85,B 0,C 180,E1 -1256.611,E2 -1256.611} C_VEL
LIN {X 0,Y 594.425,Z 485.439,A -85,B 0,C 180,E1 -1259.323,E2 -1259.323} C_VEL
LIN {X 0,Y 594.388,Z 485.439,A -85,B 0,C 180,E1 -1262.033,E2 -1262.033} C_VEL
LIN {X 0,Y 594.399,Z 485.443,A -85,B 0,C 180,E1 -1264.748,E2 -1264.748} C_VEL
LIN {X 0,Y 594.413,Z 485.439,A -85,B 0,C 180,E1 -1267.473,E2 -1267.473} C_VEL
LIN {X 0,Y 594.388,Z 485.439,A -85,B 0,C 180,E1 -1270.216,E2 -1270.216} C_VEL
LIN {X 0,Y 594.37,Z 485.451,A -85,B 0,C 180,E1 -1272.983,E2 -1272.983} C_VEL
LIN {X 0,Y 594.361,Z 485.447,A -85,B 0,C 180,E1 -1275.34,E2 -1275.34} C_VEL
LIN {X 0,Y 593.69,Z 485.527,A -85,B 0,C 180,E1 -1275.906,E2 -1275.906} C_VEL
LIN {X 0,Y 590.835,Z 485.886,A -85,B 0,C 180,E1 -1276.824,E2 -1276.824} C_VEL
LIN {X 0,Y 588.429,Z 486.184,A -85,B 0,C 180,E1 -1277.563,E2 -1277.563} C_VEL
LIN {X 0,Y 587.402,Z 486.309,A -85,B 0,C 180,E1 -1278.133,E2 -1278.133} C_VEL
LIN {X 0,Y 587.322,Z 486.32,A -85,B 0,C 180,E1 -1278.326,E2 -1278.326} C_VEL
LIN {X 0,Y 587.349,Z 486.327,A -85,B 0,C 180,E1 -1281.046,E2 -1281.046} C_VEL
LIN {X 0,Y 587.331,Z 486.317,A -85,B 0,C 180,E1 -1284.007,E2 -1284.007} C_VEL
LIN {X 0,Y 587.359,Z 486.315,A -85,B 0,C 180,E1 -1286.278,E2 -1286.278} C_VEL
LIN {X 0,Y 587.349,Z 486.324,A -85,B 0,C 180,E1 -1289.136,E2 -1289.136} C_VEL
LIN {X 0,Y 587.351,Z 486.316,A -85,B 0,C 180,E1 -1291.839,E2 -1291.839} C_VEL
LIN {X 0,Y 587.354,Z 486.316,A -85,B 0,C 180,E1 -1294.351,E2 -1294.351} C_VEL
LIN {X 0,Y 587.35,Z 486.322,A -85,B 0,C 180,E1 -1296.747,E2 -1296.747} C_VEL
LIN {X 0,Y 587.345,Z 486.321,A -85,B 0,C 180,E1 -1299.36,E2 -1299.36} C_VEL
LIN {X 0,Y 587.331,Z 486.319,A -85,B 0,C 180,E1 -1302.109,E2 -1302.109} C_VEL
LIN {X 0,Y 587.314,Z 486.33,A -85,B 0,C 180,E1 -1305.09,E2 -1305.09} C_VEL
LIN {X 0,Y 587.351,Z 486.316,A -85,B 0,C 180,E1 -1307.929,E2 -1307.929} C_VEL
LIN {X 0,Y 587.336,Z 486.327,A -85,B 0,C 180,E1 -1311.059,E2 -1311.059} C_VEL
LIN {X 0,Y 587.348,Z 486.322,A -85,B 0,C 180,E1 -1313.293,E2 -1313.293} C_VEL
LIN {X 0,Y 587.363,Z 486.315,A -85,B 0,C 180,E1 -1315.781,E2 -1315.781} C_VEL
LIN {X 0,Y 587.348,Z 486.316,A -85,B 0,C 180,E1 -1318.232,E2 -1318.232} C_VEL
LIN {X 0,Y 587.351,Z 486.325,A -85,B 0,C 180,E1 -1320.868,E2 -1320.868} C_VEL
LIN {X 0,Y 587.359,Z 486.317,A -85,B 0,C 180,E1 -1323.82,E2 -1323.82} C_VEL
LIN {X 0,Y 587.376,Z 486.333,A -85,B 0,C 180,E1 -1325.747,E2 -1325.747} C_VEL
LIN {X 0,Y 587.761,Z 491.718,A -85,B 0,C 180,E1 -1326.574,E2 -1326.574} C_VEL
LIN {X 0,Y 587.619,Z 510.319,A -85,B 0,C 180,E1 -1329.34,E2 -1329.34} C_VEL
LIN {X 0,Y 587.486,Z 530.124,A -85,B 0,C 180,E1 -1332.239,E2 -1332.239} C_VEL
LIN {X 0,Y 587.391,Z 546.111,A -85,B 0,C 180,E1 -1334.55,E2 -1334.55} C_VEL
LIN {X 0,Y 587.86,Z 550.565,A -85,B 0,C 180,E1 -1334.618,E2 -1334.618} C_VEL
LIN {X 0,Y 587.731,Z 654.423,A -85,B 0,C 180,E1 -1335.909,E2 -1335.909} C_VEL
LIN {X 0,Y 587.674,Z 668.039,A -85,B 0,C 180,E1 -1336.228,E2 -1336.228} C_VEL
LIN {X 0,Y 587.61,Z 681.098,A -85,B 0,C 180,E1 -1336.689,E2 -1336.689} C_VEL
LIN {X 0,Y 587.541,Z 692.187,A -85,B 0,C 180,E1 -1337.215,E2 -1337.215} C_VEL
LIN {X 0,Y 587.437,Z 703.708,A -85,B 0,C 180,E1 -1337.915,E2 -1337.915} C_VEL
LIN {X 0,Y 587.377,Z 714.535,A -85,B 0,C 180,E1 -1338.741,E2 -1338.741} C_VEL
LIN {X 0,Y 587.337,Z 724.211,A -85,B 0,C 180,E1 -1339.66,E2 -1339.66} C_VEL
LIN {X 0,Y 587.272,Z 733.074,A -85,B 0,C 180,E1 -1340.703,E2 -1340.703} C_VEL
LIN {X 0,Y 587.232,Z 740.176,A -85,B 0,C 180,E1 -1341.743,E2 -1341.743} C_VEL
LIN {X 0,Y 587.215,Z 745.835,A -85,B 0,C 180,E1 -1342.781,E2 -1342.781} C_VEL
LIN {X 0,Y 587.168,Z 750.282,A -85,B 0,C 180,E1 -1343.816,E2 -1343.816} C_VEL
LIN {X 0,Y 587.191,Z 752.624,A -85,B 0,C 180,E1 -1344.506,E2 -1344.506} C_VEL
LIN {X 0,Y 587.131,Z 754.535,A -85,B 0,C 180,E1 -1345.194,E2 -1345.194} C_VEL
LIN {X 0,Y 587.171,Z 756.026,A -85,B 0,C 180,E1 -1345.882,E2 -1345.882} C_VEL
LIN {X 0,Y 587.181,Z 757.065,A -85,B 0,C 180,E1 -1346.569,E2 -1346.569} C_VEL
LIN {X 0,Y 587.14,Z 757.983,A -85,B 0,C 180,E1 -1347.942,E2 -1347.942} C_VEL
LIN {X 0,Y 587.147,Z 757.853,A -85,B 0,C 180,E1 -1348.628,E2 -1348.628} C_VEL
LIN {X 0,Y 587.139,Z 756.365,A -85,B 0,C 180,E1 -1350,E2 -1350} C_VEL
LIN {X 0,Y 587.14,Z 755.04,A -85,B 0,C 180,E1 -1350.686,E2 -1350.686} C_VEL
LIN {X 0,Y 587.18,Z 752.223,A -85,B 0,C 180,E1 -1351.715,E2 -1351.715} C_VEL
LIN {X 0,Y 587.153,Z 748.396,A -85,B 0,C 180,E1 -1352.744,E2 -1352.744} C_VEL
LIN {X 0,Y 587.214,Z 743.45,A -85,B 0,C 180,E1 -1353.774,E2 -1353.774} C_VEL
LIN {X 0,Y 587.28,Z 737.238,A -85,B 0,C 180,E1 -1354.805,E2 -1354.805} C_VEL
LIN {X 0,Y 587.266,Z 729.486,A -85,B 0,C 180,E1 -1355.838,E2 -1355.838} C_VEL
LIN {X 0,Y 587.336,Z 719.813,A -85,B 0,C 180,E1 -1356.872,E2 -1356.872} C_VEL
LIN {X 0,Y 587.413,Z 709.772,A -85,B 0,C 180,E1 -1357.735,E2 -1357.735} C_VEL
LIN {X 0,Y 587.493,Z 698.471,A -85,B 0,C 180,E1 -1358.513,E2 -1358.513} C_VEL
LIN {X 0,Y 587.564,Z 687.377,A -85,B 0,C 180,E1 -1359.119,E2 -1359.119} C_VEL
LIN {X 0,Y 587.669,Z 674.938,A -85,B 0,C 180,E1 -1359.638,E2 -1359.638} C_VEL
LIN {X 0,Y 587.677,Z 661.746,A -85,B 0,C 180,E1 -1360.029,E2 -1360.029} C_VEL
LIN {X 0,Y 587.756,Z 648.812,A -85,B 0,C 180,E1 -1360.267,E2 -1360.267} C_VEL
LIN {X 0,Y 587.737,Z 548.322,A -85,B 0,C 180,E1 -1361.502,E2 -1361.502} C_VEL
LIN {X 0,Y 587.402,Z 545.998,A -85,B 0,C 180,E1 -1361.556,E2 -1361.556} C_VEL
LIN {X 0,Y 587.501,Z 526.969,A -85,B 0,C 180,E1 -1364.31,E2 -1364.31} C_VEL
LIN {X 0,Y 587.615,Z 508.082,A -85,B 0,C 180,E1 -1367.081,E2 -1367.081} C_VEL
LIN {X 0,Y 587.762,Z 490.218,A -85,B 0,C 180,E1 -1369.742,E2 -1369.742} C_VEL
LIN {X 0,Y 587.337,Z 486.325,A -85,B 0,C 180,E1 -1370.35,E2 -1370.35} C_VEL
LIN {X 0,Y 587.317,Z 486.329,A -85,B 0,C 180,E1 -1373.258,E2 -1373.258} C_VEL
LIN {X 0,Y 587.333,Z 486.322,A -85,B 0,C 180,E1 -1375.516,E2 -1375.516} C_VEL
LIN {X 0,Y 587.349,Z 486.317,A -85,B 0,C 180,E1 -1377.817,E2 -1377.817} C_VEL
LIN {X 0,Y 587.345,Z 486.32,A -85,B 0,C 180,E1 -1380.51,E2 -1380.51} C_VEL
LIN {X 0,Y 587.339,Z 486.326,A -85,B 0,C 180,E1 -1383.111,E2 -1383.111} C_VEL
LIN {X 0,Y 587.298,Z 486.325,A -85,B 0,C 180,E1 -1385.537,E2 -1385.537} C_VEL
LIN {X 0,Y 587.343,Z 486.317,A -85,B 0,C 180,E1 -1387.838,E2 -1387.838} C_VEL
LIN {X 0,Y 587.32,Z 486.321,A -85,B 0,C 180,E1 -1390.253,E2 -1390.253} C_VEL
LIN {X 0,Y 587.336,Z 486.324,A -85,B 0,C 180,E1 -1393.12,E2 -1393.12} C_VEL
LIN {X 0,Y 587.332,Z 486.318,A -85,B 0,C 180,E1 -1396.05,E2 -1396.05} C_VEL
LIN {X 0,Y 587.334,Z 486.327,A -85,B 0,C 180,E1 -1398.924,E2 -1398.924} C_VEL
LIN {X 0,Y 587.328,Z 486.32,A -85,B 0,C 180,E1 -1401.52,E2 -1401.52} C_VEL
LIN {X 0,Y 587.349,Z 486.322,A -85,B 0,C 180,E1 -1404.453,E2 -1404.453} C_VEL
LIN {X 0,Y 587.335,Z 486.327,A -85,B 0,C 180,E1 -1406.887,E2 -1406.887} C_VEL
LIN {X 0,Y 587.372,Z 486.471,A -85,B 0,C 180,E1 -1408.158,E2 -1408.158} C_VEL
LIN {X 0,Y 587.302,Z 498.353,A -85,B 0,C 180,E1 -1410.568,E2 -1410.568} C_VEL
LIN {X 0,Y 587.865,Z 503.02,A -85,B 0,C 180,E1 -1410.649,E2 -1410.649} C_VEL
LIN {X 0,Y 587.712,Z 604.406,A -85,B 0,C 180,E1 -1411.91,E2 -1411.91} C_VEL
LIN {X 0,Y 587.654,Z 617.791,A -85,B 0,C 180,E1 -1412.221,E2 -1412.221} C_VEL
LIN {X 0,Y 587.598,Z 630.815,A -85,B 0,C 180,E1 -1412.678,E2 -1412.678} C_VEL
LIN {X 0,Y 587.509,Z 642.78,A -85,B 0,C 180,E1 -1413.251,E2 -1413.251} C_VEL
LIN {X 0,Y 587.438,Z 653.716,A -85,B 0,C 180,E1 -1413.917,E2 -1413.917} C_VEL
LIN {X 0,Y 587.383,Z 664.883,A -85,B 0,C 180,E1 -1414.77,E2 -1414.77} C_VEL
LIN {X 0,Y 587.3,Z 674.173,A -85,B 0,C 180,E1 -1415.657,E2 -1415.657} C_VEL
LIN {X 0,Y 587.268,Z 681.885,A -85,B 0,C 180,E1 -1416.552,E2 -1416.552} C_VEL
LIN {X 0,Y 587.21,Z 688.493,A -85,B 0,C 180,E1 -1417.481,E2 -1417.481} C_VEL
LIN {X 0,Y 587.213,Z 694.867,A -85,B 0,C 180,E1 -1418.59,E2 -1418.59} C_VEL
LIN {X 0,Y 587.193,Z 699.803,A -85,B 0,C 180,E1 -1419.69,E2 -1419.69} C_VEL
LIN {X 0,Y 587.151,Z 704.066,A -85,B 0,C 180,E1 -1421.011,E2 -1421.011} C_VEL
LIN {X 0,Y 587.126,Z 706,A -85,B 0,C 180,E1 -1421.867,E2 -1421.867} C_VEL
LIN {X 0,Y 587.126,Z 707.09,A -85,B 0,C 180,E1 -1422.587,E2 -1422.587} C_VEL
LIN {X 0,Y 587.153,Z 707.741,A -85,B 0,C 180,E1 -1423.305,E2 -1423.305} C_VEL
LIN {X 0,Y 587.155,Z 707.998,A -85,B 0,C 180,E1 -1424.02,E2 -1424.02} C_VEL
LIN {X 0,Y 587.14,Z 707.789,A -85,B 0,C 180,E1 -1424.732,E2 -1424.732} C_VEL
LIN {X 0,Y 587.174,Z 706.129,A -85,B 0,C 180,E1 -1426.15,E2 -1426.15} C_VEL
LIN {X 0,Y 587.142,Z 704.651,A -85,B 0,C 180,E1 -1426.854,E2 -1426.854} C_VEL
LIN {X 0,Y 587.168,Z 701.595,A -85,B 0,C 180,E1 -1427.909,E2 -1427.909} C_VEL
LIN {X 0,Y 587.19,Z 697.473,A -85,B 0,C 180,E1 -1428.959,E2 -1428.959} C_VEL
LIN {X 0,Y 587.195,Z 691.151,A -85,B 0,C 180,E1 -1430.18,E2 -1430.18} C_VEL
LIN {X 0,Y 587.277,Z 684.267,A -85,B 0,C 180,E1 -1431.223,E2 -1431.223} C_VEL
LIN {X 0,Y 587.275,Z 675.787,A -85,B 0,C 180,E1 -1432.263,E2 -1432.263} C_VEL
LIN {X 0,Y 587.384,Z 665.707,A -85,B 0,C 180,E1 -1433.248,E2 -1433.248} C_VEL
LIN {X 0,Y 587.439,Z 656.337,A -85,B 0,C 180,E1 -1433.991,E2 -1433.991} C_VEL
LIN {X 0,Y 587.494,Z 645.635,A -85,B 0,C 180,E1 -1434.68,E2 -1434.68} C_VEL
LIN {X 0,Y 587.579,Z 633.799,A -85,B 0,C 180,E1 -1435.283,E2 -1435.283} C_VEL
LIN {X 0,Y 587.662,Z 621.471,A -85,B 0,C 180,E1 -1435.756,E2 -1435.756} C_VEL
LIN {X 0,Y 587.736,Z 608.601,A -85,B 0,C 180,E1 -1436.1,E2 -1436.1} C_VEL
LIN {X 0,Y 587.755,Z 593.251,A -85,B 0,C 180,E1 -1436.336,E2 -1436.336} C_VEL
LIN {X 0,Y 587.818,Z 501.421,A -85,B 0,C 180,E1 -1437.462,E2 -1437.462} C_VEL
LIN {X 0,Y 587.289,Z 498.394,A -85,B 0,C 180,E1 -1437.514,E2 -1437.514} C_VEL
LIN {X 0,Y 587.37,Z 486.317,A -85,B 0,C 180,E1 -1440,E2 -1440} C_VEL
LIN {X 0,Y 587.376,Z 486.316,A -85,B 0,C 180,E1 -1442.743,E2 -1442.743} C_VEL
LIN {X 0,Y 587.363,Z 486.323,A -85,B 0,C 180,E1 -1445.493,E2 -1445.493} C_VEL
LIN {X 0,Y 587.365,Z 486.315,A -85,B 0,C 180,E1 -1448.255,E2 -1448.255} C_VEL
LIN {X 0,Y 587.352,Z 486.325,A -85,B 0,C 180,E1 -1451.141,E2 -1451.141} C_VEL
LIN {X 0,Y 587.355,Z 486.316,A -85,B 0,C 180,E1 -1454.261,E2 -1454.261} C_VEL
LIN {X 0,Y 587.354,Z 486.323,A -85,B 0,C 180,E1 -1457.406,E2 -1457.406} C_VEL
LIN {X 0,Y 587.328,Z 486.319,A -85,B 0,C 180,E1 -1460.305,E2 -1460.305} C_VEL
LIN {X 0,Y 587.316,Z 486.329,A -85,B 0,C 180,E1 -1463.259,E2 -1463.259} C_VEL
LIN {X 0,Y 587.356,Z 486.315,A -85,B 0,C 180,E1 -1466.183,E2 -1466.183} C_VEL
LIN {X 0,Y 587.347,Z 486.326,A -85,B 0,C 180,E1 -1469.135,E2 -1469.135} C_VEL
LIN {X 0,Y 587.349,Z 486.317,A -85,B 0,C 180,E1 -1471.838,E2 -1471.838} C_VEL
LIN {X 0,Y 587.353,Z 486.316,A -85,B 0,C 180,E1 -1474.35,E2 -1474.35} C_VEL
LIN {X 0,Y 587.348,Z 486.321,A -85,B 0,C 180,E1 -1476.747,E2 -1476.747} C_VEL
LIN {X 0,Y 587.343,Z 486.322,A -85,B 0,C 180,E1 -1479.36,E2 -1479.36} C_VEL
LIN {X 0,Y 587.329,Z 486.319,A -85,B 0,C 180,E1 -1482.109,E2 -1482.109} C_VEL
LIN {X 0,Y 587.312,Z 486.33,A -85,B 0,C 180,E1 -1485.09,E2 -1485.09} C_VEL
LIN {X 0,Y 587.349,Z 486.317,A -85,B 0,C 180,E1 -1487.928,E2 -1487.928} C_VEL
LIN {X 0,Y 587.332,Z 486.327,A -85,B 0,C 180,E1 -1491.059,E2 -1491.059} C_VEL
LIN {X 0,Y 587.35,Z 486.321,A -85,B 0,C 180,E1 -1493.293,E2 -1493.293} C_VEL
LIN {X 0,Y 587.359,Z 486.316,A -85,B 0,C 180,E1 -1495.781,E2 -1495.781} C_VEL
LIN {X 0,Y 587.351,Z 486.319,A -85,B 0,C 180,E1 -1498.233,E2 -1498.233} C_VEL
LIN {X 0,Y 587.348,Z 486.327,A -85,B 0,C 180,E1 -1500.867,E2 -1500.867} C_VEL
LIN {X 0,Y 587.357,Z 486.317,A -85,B 0,C 180,E1 -1503.82,E2 -1503.82} C_VEL
LIN {X 0,Y 587.336,Z 486.401,A -85,B 0,C 180,E1 -1505.273,E2 -1505.273} C_VEL
LIN {X 0,Y 588.06,Z 490.63,A -85,B 0,C 180,E1 -1505.86,E2 -1505.86} C_VEL
LIN {X 0,Y 587.897,Z 512.128,A -85,B 0,C 180,E1 -1508.635,E2 -1508.635} C_VEL
LIN {X 0,Y 587.722,Z 536.383,A -85,B 0,C 180,E1 -1511.706,E2 -1511.706} C_VEL
LIN {X 0,Y 587.525,Z 560.778,A -85,B 0,C 180,E1 -1514.742,E2 -1514.742} C_VEL
LIN {X 0,Y 587.504,Z 575.275,A -85,B 0,C 180,E1 -1516.5,E2 -1516.5} C_VEL
LIN {X 0,Y 587.871,Z 579.746,A -85,B 0,C 180,E1 -1516.563,E2 -1516.563} C_VEL
LIN {X 0,Y 587.717,Z 683.961,A -85,B 0,C 180,E1 -1517.855,E2 -1517.855} C_VEL
LIN {X 0,Y 587.666,Z 697.224,A -85,B 0,C 180,E1 -1518.161,E2 -1518.161} C_VEL
LIN {X 0,Y 587.608,Z 709.77,A -85,B 0,C 180,E1 -1518.59,E2 -1518.59} C_VEL
LIN {X 0,Y 587.554,Z 721.637,A -85,B 0,C 180,E1 -1519.141,E2 -1519.141} C_VEL
LIN {X 0,Y 587.458,Z 733.205,A -85,B 0,C 180,E1 -1519.837,E2 -1519.837} C_VEL
LIN {X 0,Y 587.391,Z 743.6,A -85,B 0,C 180,E1 -1520.618,E2 -1520.618} C_VEL
LIN {X 0,Y 587.321,Z 752.114,A -85,B 0,C 180,E1 -1521.398,E2 -1521.398} C_VEL
LIN {X 0,Y 587.273,Z 759.962,A -85,B 0,C 180,E1 -1522.263,E2 -1522.263} C_VEL
LIN {X 0,Y 587.23,Z 766.471,A -85,B 0,C 180,E1 -1523.127,E2 -1523.127} C_VEL
LIN {X 0,Y 587.236,Z 772.867,A -85,B 0,C 180,E1 -1524.161,E2 -1524.161} C_VEL
LIN {X 0,Y 587.147,Z 777.95,A -85,B 0,C 180,E1 -1525.194,E2 -1525.194} C_VEL
LIN {X 0,Y 587.212,Z 781.896,A -85,B 0,C 180,E1 -1526.226,E2 -1526.226} C_VEL
LIN {X 0,Y 587.132,Z 784.81,A -85,B 0,C 180,E1 -1527.256,E2 -1527.256} C_VEL
LIN {X 0,Y 587.138,Z 786.201,A -85,B 0,C 180,E1 -1527.942,E2 -1527.942} C_VEL
LIN {X 0,Y 587.14,Z 787.784,A -85,B 0,C 180,E1 -1529.314,E2 -1529.314} C_VEL
LIN {X 0,Y 587.137,Z 788,A -85,B 0,C 180,E1 -1530,E2 -1530} C_VEL
LIN {X 0,Y 587.147,Z 787.185,A -85,B 0,C 180,E1 -1531.372,E2 -1531.372} C_VEL
LIN {X 0,Y 587.138,Z 786.201,A -85,B 0,C 180,E1 -1532.058,E2 -1532.058} C_VEL
LIN {X 0,Y 587.132,Z 784.809,A -85,B 0,C 180,E1 -1532.744,E2 -1532.744} C_VEL
LIN {X 0,Y 587.212,Z 781.896,A -85,B 0,C 180,E1 -1533.774,E2 -1533.774} C_VEL
LIN {X 0,Y 587.147,Z 777.95,A -85,B 0,C 180,E1 -1534.806,E2 -1534.806} C_VEL
LIN {X 0,Y 587.217,Z 771.878,A -85,B 0,C 180,E1 -1536.011,E2 -1536.011} C_VEL
LIN {X 0,Y 587.245,Z 765.238,A -85,B 0,C 180,E1 -1537.046,E2 -1537.046} C_VEL
LIN {X 0,Y 587.299,Z 756.992,A -85,B 0,C 180,E1 -1538.083,E2 -1538.083} C_VEL
LIN {X 0,Y 587.343,Z 748.54,A -85,B 0,C 180,E1 -1538.949,E2 -1538.949} C_VEL
LIN {X 0,Y 587.41,Z 738.098,A -85,B 0,C 180,E1 -1539.816,E2 -1539.816} C_VEL
LIN {X 0,Y 587.505,Z 727.762,A -85,B 0,C 180,E1 -1540.511,E2 -1540.511} C_VEL
LIN {X 0,Y 587.583,Z 715.806,A -85,B 0,C 180,E1 -1541.149,E2 -1541.149} C_VEL
LIN {X 0,Y 587.624,Z 703.602,A -85,B 0,C 180,E1 -1541.639,E2 -1541.639} C_VEL
LIN {X 0,Y 587.669,Z 690.451,A -85,B 0,C 180,E1 -1542.014,E2 -1542.014} C_VEL
LIN {X 0,Y 587.771,Z 678.106,A -85,B 0,C 180,E1 -1542.231,E2 -1542.231} C_VEL
LIN {X 0,Y 587.757,Z 577.176,A -85,B 0,C 180,E1 -1543.471,E2 -1543.471} C_VEL
LIN {X 0,Y 587.473,Z 574.948,A -85,B 0,C 180,E1 -1543.512,E2 -1543.512} C_VEL
LIN {X 0,Y 587.595,Z 550.733,A -85,B 0,C 180,E1 -1546.503,E2 -1546.503} C_VEL
LIN {X 0,Y 587.744,Z 528.446,A -85,B 0,C 180,E1 -1549.294,E2 -1549.294} C_VEL
LIN {X 0,Y 587.946,Z 506.248,A -85,B 0,C 180,E1 -1552.119,E2 -1552.119} C_VEL
LIN {X 0,Y 587.992,Z 489.363,A -85,B 0,C 180,E1 -1554.309,E2 -1554.309} C_VEL
LIN {X 0,Y 587.314,Z 486.329,A -85,B 0,C 180,E1 -1554.76,E2 -1554.76} C_VEL
LIN {X 0,Y 587.33,Z 486.328,A -85,B 0,C 180,E1 -1557.045,E2 -1557.045} C_VEL
LIN {X 0,Y 587.345,Z 486.325,A -85,B 0,C 180,E1 -1559.379,E2 -1559.379} C_VEL
LIN {X 0,Y 587.353,Z 486.317,A -85,B 0,C 180,E1 -1561.837,E2 -1561.837} C_VEL
LIN {X 0,Y 587.345,Z 486.317,A -85,B 0,C 180,E1 -1564.347,E2 -1564.347} C_VEL
LIN {X 0,Y 587.344,Z 486.318,A -85,B 0,C 180,E1 -1567.607,E2 -1567.607} C_VEL
LIN {X 0,Y 587.316,Z 486.32,A -85,B 0,C 180,E1 -1570.253,E2 -1570.253} C_VEL
LIN {X 0,Y 587.323,Z 486.329,A -85,B 0,C 180,E1 -1573.119,E2 -1573.119} C_VEL
LIN {X 0,Y 587.317,Z 486.321,A -85,B 0,C 180,E1 -1576.049,E2 -1576.049} C_VEL
LIN {X 0,Y 587.331,Z 486.324,A -85,B 0,C 180,E1 -1578.924,E2 -1578.924} C_VEL
LIN {X 0,Y 587.326,Z 486.323,A -85,B 0,C 180,E1 -1581.52,E2 -1581.52} C_VEL
LIN {X 0,Y 587.348,Z 486.316,A -85,B 0,C 180,E1 -1584.453,E2 -1584.453} C_VEL
LIN {X 0,Y 587.333,Z 486.324,A -85,B 0,C 180,E1 -1586.887,E2 -1586.887} C_VEL
LIN {X 0,Y 587.343,Z 486.321,A -85,B 0,C 180,E1 -1589.487,E2 -1589.487} C_VEL
LIN {X 0,Y 587.343,Z 486.317,A -85,B 0,C 180,E1 -1592.306,E2 -1592.306} C_VEL
LIN {X 0,Y 587.334,Z 486.319,A -85,B 0,C 180,E1 -1594.483,E2 -1594.483} C_VEL
LIN {X 0,Y 587.333,Z 486.322,A -85,B 0,C 180,E1 -1597.486,E2 -1597.486} C_VEL
LIN {X 0,Y 587.327,Z 486.321,A -85,B 0,C 180,E1 -1599.695,E2 -1599.695} C_VEL
LIN {X 0,Y 587.35,Z 486.317,A -85,B 0,C 180,E1 -1602.594,E2 -1602.594} C_VEL
LIN {X 0,Y 587.354,Z 486.317,A -85,B 0,C 180,E1 -1605.739,E2 -1605.739} C_VEL
LIN {X 0,Y 587.352,Z 486.322,A -85,B 0,C 180,E1 -1608.859,E2 -1608.859} C_VEL
LIN {X 0,Y 587.364,Z 486.314,A -85,B 0,C 180,E1 -1611.745,E2 -1611.745} C_VEL
LIN {X 0,Y 587.357,Z 486.316,A -85,B 0,C 180,E1 -1614.507,E2 -1614.507} C_VEL
LIN {X 0,Y 587.377,Z 486.32,A -85,B 0,C 180,E1 -1617.257,E2 -1617.257} C_VEL
LIN {X 0,Y 587.373,Z 486.311,A -85,B 0,C 180,E1 -1620,E2 -1620} C_VEL
LIN {X 0,Y 587.376,Z 486.317,A -85,B 0,C 180,E1 -1622.743,E2 -1622.743} C_VEL
LIN {X 0,Y 587.362,Z 486.318,A -85,B 0,C 180,E1 -1625.493,E2 -1625.493} C_VEL
LIN {X 0,Y 587.364,Z 486.312,A -85,B 0,C 180,E1 -1628.255,E2 -1628.255} C_VEL
LIN {X 0,Y 587.352,Z 486.325,A -85,B 0,C 180,E1 -1631.142,E2 -1631.142} C_VEL
LIN {X 0,Y 587.355,Z 486.315,A -85,B 0,C 180,E1 -1634.261,E2 -1634.261} C_VEL
LIN {X 0,Y 587.353,Z 486.32,A -85,B 0,C 180,E1 -1637.406,E2 -1637.406} C_VEL
LIN {X 0,Y 587.322,Z 486.32,A -85,B 0,C 180,E1 -1638.326,E2 -1638.326} C_VEL
LIN {X 0,Y 586.669,Z 486.409,A -85,B 0,C 180,E1 -1638.898,E2 -1638.898} C_VEL
LIN {X 0,Y 583.837,Z 486.765,A -85,B 0,C 180,E1 -1639.826,E2 -1639.826} C_VEL
LIN {X 0,Y 581.427,Z 487.066,A -85,B 0,C 180,E1 -1640.573,E2 -1640.573} C_VEL
LIN {X 0,Y 580.374,Z 487.193,A -85,B 0,C 180,E1 -1641.149,E2 -1641.149} C_VEL
LIN {X 0,Y 580.279,Z 487.202,A -85,B 0,C 180,E1 -1641.345,E2 -1641.345} C_VEL
LIN {X 0,Y 580.294,Z 487.194,A -85,B 0,C 180,E1 -1644.317,E2 -1644.317} C_VEL
LIN {X 0,Y 580.305,Z 487.197,A -85,B 0,C 180,E1 -1646.622,E2 -1646.622} C_VEL
LIN {X 0,Y 580.302,Z 487.199,A -85,B 0,C 180,E1 -1649.312,E2 -1649.312} C_VEL
LIN {X 0,Y 580.298,Z 487.195,A -85,B 0,C 180,E1 -1652.201,E2 -1652.201} C_VEL
LIN {X 0,Y 580.299,Z 487.199,A -85,B 0,C 180,E1 -1654.696,E2 -1654.696} C_VEL
LIN {X 0,Y 580.297,Z 487.201,A -85,B 0,C 180,E1 -1657.269,E2 -1657.269} C_VEL
LIN {X 0,Y 580.295,Z 487.195,A -85,B 0,C 180,E1 -1660.273,E2 -1660.273} C_VEL
LIN {X 0,Y 580.278,Z 487.203,A -85,B 0,C 180,E1 -1662.707,E2 -1662.707} C_VEL
LIN {X 0,Y 580.272,Z 487.2,A -85,B 0,C 180,E1 -1665.61,E2 -1665.61} C_VEL
LIN {X 0,Y 580.313,Z 487.193,A -85,B 0,C 180,E1 -1668.235,E2 -1668.235} C_VEL
LIN {X 0,Y 580.291,Z 487.206,A -85,B 0,C 180,E1 -1670.967,E2 -1670.967} C_VEL
LIN {X 0,Y 580.269,Z 487.2,A -85,B 0,C 180,E1 -1673.597,E2 -1673.597} C_VEL
LIN {X 0,Y 580.317,Z 487.193,A -85,B 0,C 180,E1 -1676.146,E2 -1676.146} C_VEL
LIN {X 0,Y 580.284,Z 487.2,A -85,B 0,C 180,E1 -1678.616,E2 -1678.616} C_VEL
LIN {X 0,Y 580.294,Z 487.206,A -85,B 0,C 180,E1 -1681.025,E2 -1681.025} C_VEL
LIN {X 0,Y 580.293,Z 487.198,A -85,B 0,C 180,E1 -1683.667,E2 -1683.667} C_VEL
LIN {X 0,Y 580.369,Z 487.388,A -85,B 0,C 180,E1 -1685.624,E2 -1685.624} C_VEL
LIN {X 0,Y 580.818,Z 491.538,A -85,B 0,C 180,E1 -1686.277,E2 -1686.277} C_VEL
LIN {X 0,Y 580.655,Z 508.606,A -85,B 0,C 180,E1 -1688.851,E2 -1688.851} C_VEL
LIN {X 0,Y 580.526,Z 526.238,A -85,B 0,C 180,E1 -1691.471,E2 -1691.471} C_VEL
LIN {X 0,Y 580.379,Z 546.153,A -85,B 0,C 180,E1 -1694.387,E2 -1694.387} C_VEL
LIN {X 0,Y 580.965,Z 550.381,A -85,B 0,C 180,E1 -1694.454,E2 -1694.454} C_VEL
LIN {X 0,Y 580.806,Z 654.702,A -85,B 0,C 180,E1 -1695.767,E2 -1695.767} C_VEL
LIN {X 0,Y 580.73,Z 667.968,A -85,B 0,C 180,E1 -1696.083,E2 -1696.083} C_VEL
LIN {X 0,Y 580.672,Z 680.507,A -85,B 0,C 180,E1 -1696.527,E2 -1696.527} C_VEL
LIN {X 0,Y 580.556,Z 691.727,A -85,B 0,C 180,E1 -1697.059,E2 -1697.059} C_VEL
LIN {X 0,Y 580.429,Z 703.356,A -85,B 0,C 180,E1 -1697.767,E2 -1697.767} C_VEL
LIN {X 0,Y 580.348,Z 713.883,A -85,B 0,C 180,E1 -1698.572,E2 -1698.572} C_VEL
LIN {X 0,Y 580.306,Z 722.424,A -85,B 0,C 180,E1 -1699.37,E2 -1699.37} C_VEL
LIN {X 0,Y 580.201,Z 731.532,A -85,B 0,C 180,E1 -1700.413,E2 -1700.413} C_VEL
LIN {X 0,Y 580.161,Z 738.935,A -85,B 0,C 180,E1 -1701.466,E2 -1701.466} C_VEL
LIN {X 0,Y 580.126,Z 745.724,A -85,B 0,C 180,E1 -1702.692,E2 -1702.692} C_VEL
LIN {X 0,Y 580.084,Z 750.197,A -85,B 0,C 180,E1 -1703.74,E2 -1703.74} C_VEL
LIN {X 0,Y 580.112,Z 752.552,A -85,B 0,C 180,E1 -1704.438,E2 -1704.438} C_VEL
LIN {X 0,Y 580.035,Z 754.474,A -85,B 0,C 180,E1 -1705.135,E2 -1705.135} C_VEL
LIN {X 0,Y 580.088,Z 755.981,A -85,B 0,C 180,E1 -1705.831,E2 -1705.831} C_VEL
LIN {X 0,Y 580.107,Z 757.038,A -85,B 0,C 180,E1 -1706.527,E2 -1706.527} C_VEL
LIN {X 0,Y 580.039,Z 757.977,A -85,B 0,C 180,E1 -1707.917,E2 -1707.917} C_VEL
LIN {X 0,Y 580.046,Z 757.867,A -85,B 0,C 180,E1 -1708.611,E2 -1708.611} C_VEL
LIN {X 0,Y 580.04,Z 756.403,A -85,B 0,C 180,E1 -1710,E2 -1710} C_VEL
LIN {X 0,Y 580.041,Z 755.089,A -85,B 0,C 180,E1 -1710.694,E2 -1710.694} C_VEL
LIN {X 0,Y 580.086,Z 752.297,A -85,B 0,C 180,E1 -1711.736,E2 -1711.736} C_VEL
LIN {X 0,Y 580.066,Z 748.496,A -85,B 0,C 180,E1 -1712.778,E2 -1712.778} C_VEL
LIN {X 0,Y 580.141,Z 743.576,A -85,B 0,C 180,E1 -1713.82,E2 -1713.82} C_VEL
LIN {X 0,Y 580.206,Z 737.394,A -85,B 0,C 180,E1 -1714.864,E2 -1714.864} C_VEL
LIN {X 0,Y 580.209,Z 729.682,A -85,B 0,C 180,E1 -1715.909,E2 -1715.909} C_VEL
LIN {X 0,Y 580.316,Z 721.353,A -85,B 0,C 180,E1 -1716.828,E2 -1716.828} C_VEL
LIN {X 0,Y 580.389,Z 711.188,A -85,B 0,C 180,E1 -1717.742,E2 -1717.742} C_VEL
LIN {X 0,Y 580.486,Z 700.255,A -85,B 0,C 180,E1 -1718.529,E2 -1718.529} C_VEL
LIN {X 0,Y 580.613,Z 689.598,A -85,B 0,C 180,E1 -1719.141,E2 -1719.141} C_VEL
LIN {X 0,Y 580.648,Z 677.9,A -85,B 0,C 180,E1 -1719.668,E2 -1719.668} C_VEL
LIN {X 0,Y 580.734,Z 664.466,A -85,B 0,C 180,E1 -1720.106,E2 -1720.106} C_VEL
LIN {X 0,Y 580.781,Z 652.005,A -85,B 0,C 180,E1 -1720.37,E2 -1720.37} C_VEL
LIN {X 0,Y 580.814,Z 548.936,A -85,B 0,C 180,E1 -1721.658,E2 -1721.658} C_VEL
LIN {X 0,Y 580.39,Z 545.925,A -85,B 0,C 180,E1 -1721.733,E2 -1721.733} C_VEL
LIN {X 0,Y 580.535,Z 525.502,A -85,B 0,C 180,E1 -1724.727,E2 -1724.727} C_VEL
LIN {X 0,Y 580.675,Z 506.117,A -85,B 0,C 180,E1 -1727.612,E2 -1727.612} C_VEL
LIN {X 0,Y 580.836,Z 490.393,A -85,B 0,C 180,E1 -1729.987,E2 -1729.987} C_VEL
LIN {X 0,Y 580.311,Z 487.201,A -85,B 0,C 180,E1 -1730.515,E2 -1730.515} C_VEL
LIN {X 0,Y 580.275,Z 487.202,A -85,B 0,C 180,E1 -1733.558,E2 -1733.558} C_VEL
LIN {X 0,Y 580.292,Z 487.197,A -85,B 0,C 180,E1 -1735.848,E2 -1735.848} C_VEL
LIN {X 0,Y 580.301,Z 487.195,A -85,B 0,C 180,E1 -1738.185,E2 -1738.185} C_VEL
LIN {X 0,Y 580.295,Z 487.201,A -85,B 0,C 180,E1 -1740.695,E2 -1740.695} C_VEL
LIN {X 0,Y 580.304,Z 487.199,A -85,B 0,C 180,E1 -1743.315,E2 -1743.315} C_VEL
LIN {X 0,Y 580.247,Z 487.201,A -85,B 0,C 180,E1 -1745.756,E2 -1745.756} C_VEL
LIN {X 0,Y 580.29,Z 487.196,A -85,B 0,C 180,E1 -1748.145,E2 -1748.145} C_VEL
LIN {X 0,Y 580.301,Z 487.203,A -85,B 0,C 180,E1 -1750.842,E2 -1750.842} C_VEL
LIN {X 0,Y 580.289,Z 487.196,A -85,B 0,C 180,E1 -1753.656,E2 -1753.656} C_VEL
LIN {X 0,Y 580.283,Z 487.202,A -85,B 0,C 180,E1 -1756.607,E2 -1756.607} C_VEL
LIN {X 0,Y 580.297,Z 487.2,A -85,B 0,C 180,E1 -1759.156,E2 -1759.156} C_VEL
LIN {X 0,Y 580.286,Z 487.197,A -85,B 0,C 180,E1 -1761.926,E2 -1761.926} C_VEL
LIN {X 0,Y 580.304,Z 487.2,A -85,B 0,C 180,E1 -1764.456,E2 -1764.456} C_VEL
LIN {X 0,Y 580.29,Z 487.204,A -85,B 0,C 180,E1 -1766.975,E2 -1766.975} C_VEL
LIN {X 0,Y 580.346,Z 487.286,A -85,B 0,C 180,E1 -1768.129,E2 -1768.129} C_VEL
LIN {X 0,Y 580.269,Z 498.461,A -85,B 0,C 180,E1 -1770.413,E2 -1770.413} C_VEL
LIN {X 0,Y 580.978,Z 503.555,A -85,B 0,C 180,E1 -1770.493,E2 -1770.493} C_VEL
LIN {X 0,Y 580.824,Z 603.152,A -85,B 0,C 180,E1 -1771.743,E2 -1771.743} C_VEL
LIN {X 0,Y 580.753,Z 614.669,A -85,B 0,C 180,E1 -1771.992,E2 -1771.992} C_VEL
LIN {X 0,Y 580.671,Z 626.722,A -85,B 0,C 180,E1 -1772.376,E2 -1772.376} C_VEL
LIN {X 0,Y 580.544,Z 640.619,A -85,B 0,C 180,E1 -1773.001,E2 -1773.001} C_VEL
LIN {X 0,Y 580.431,Z 651.367,A -85,B 0,C 180,E1 -1773.636,E2 -1773.636} C_VEL
LIN {X 0,Y 580.37,Z 661.132,A -85,B 0,C 180,E1 -1774.347,E2 -1774.347} C_VEL
LIN {X 0,Y 580.302,Z 670.064,A -85,B 0,C 180,E1 -1775.135,E2 -1775.135} C_VEL
LIN {X 0,Y 580.213,Z 678.671,A -85,B 0,C 180,E1 -1776.06,E2 -1776.06} C_VEL
LIN {X 0,Y 580.166,Z 687.151,A -85,B 0,C 180,E1 -1777.192,E2 -1777.192} C_VEL
LIN {X 0,Y 580.134,Z 692.809,A -85,B 0,C 180,E1 -1778.129,E2 -1778.129} C_VEL
LIN {X 0,Y 580.098,Z 697.826,A -85,B 0,C 180,E1 -1779.158,E2 -1779.158} C_VEL
LIN {X 0,Y 580.086,Z 701.688,A -85,B 0,C 180,E1 -1780.17,E2 -1780.17} C_VEL
LIN {X 0,Y 580.056,Z 703.916,A -85,B 0,C 180,E1 -1780.914,E2 -1780.914} C_VEL
LIN {X 0,Y 580.034,Z 705.589,A -85,B 0,C 180,E1 -1781.637,E2 -1781.637} C_VEL
LIN {X 0,Y 580.037,Z 706.812,A -85,B 0,C 180,E1 -1782.367,E2 -1782.367} C_VEL
LIN {X 0,Y 580.029,Z 707.658,A -85,B 0,C 180,E1 -1783.175,E2 -1783.175} C_VEL
LIN {X 0,Y 580.06,Z 707.962,A -85,B 0,C 180,E1 -1783.819,E2 -1783.819} C_VEL
LIN {X 0,Y 580.035,Z 707.868,A -85,B 0,C 180,E1 -1784.54,E2 -1784.54} C_VEL
LIN {X 0,Y 580.056,Z 706.788,A -85,B 0,C 180,E1 -1785.757,E2 -1785.757} C_VEL
LIN {X 0,Y 580.06,Z 705.076,A -85,B 0,C 180,E1 -1786.691,E2 -1786.691} C_VEL
LIN {X 0,Y 580.073,Z 702.213,A -85,B 0,C 180,E1 -1787.759,E2 -1787.759} C_VEL
LIN {X 0,Y 580.101,Z 697.977,A -85,B 0,C 180,E1 -1788.902,E2 -1788.902} C_VEL
LIN {X 0,Y 580.129,Z 693.249,A -85,B 0,C 180,E1 -1789.883,E2 -1789.883} C_VEL
LIN {X 0,Y 580.15,Z 686.905,A -85,B 0,C 180,E1 -1790.939,E2 -1790.939} C_VEL
LIN {X 0,Y 580.234,Z 678.953,A -85,B 0,C 180,E1 -1791.993,E2 -1791.993} C_VEL
LIN {X 0,Y 580.3,Z 670.896,A -85,B 0,C 180,E1 -1792.869,E2 -1792.869} C_VEL
LIN {X 0,Y 580.357,Z 662.854,A -85,B 0,C 180,E1 -1793.6,E2 -1793.6} C_VEL
LIN {X 0,Y 580.411,Z 652.878,A -85,B 0,C 180,E1 -1794.354,E2 -1794.354} C_VEL
LIN {X 0,Y 580.556,Z 641.354,A -85,B 0,C 180,E1 -1795.052,E2 -1795.052} C_VEL
LIN {X 0,Y 580.655,Z 629.126,A -85,B 0,C 180,E1 -1795.618,E2 -1795.618} C_VEL
LIN {X 0,Y 580.718,Z 617.063,A -85,B 0,C 180,E1 -1796.031,E2 -1796.031} C_VEL
LIN {X 0,Y 580.797,Z 604.001,A -85,B 0,C 180,E1 -1796.336,E2 -1796.336} C_VEL
LIN {X 0,Y 580.883,Z 502.165,A -85,B 0,C 180,E1 -1797.616,E2 -1797.616} C_VEL
LIN {X 0,Y 580.262,Z 498.293,A -85,B 0,C 180,E1 -1797.7,E2 -1797.7} C_VEL
LIN {X 0,Y 580.327,Z 487.195,A -85,B 0,C 180,E1 -1800,E2 -1800} C_VEL
LIN {X 0,Y 580.341,Z 487.193,A -85,B 0,C 180,E1 -1802.776,E2 -1802.776} C_VEL
LIN {X 0,Y 580.329,Z 487.198,A -85,B 0,C 180,E1 -1805.56,E2 -1805.56} C_VEL
LIN {X 0,Y 580.328,Z 487.192,A -85,B 0,C 180,E1 -1808.356,E2 -1808.356} C_VEL
LIN {X 0,Y 580.323,Z 487.202,A -85,B 0,C 180,E1 -1811.208,E2 -1811.208} C_VEL
LIN {X 0,Y 580.318,Z 487.193,A -85,B 0,C 180,E1 -1814.017,E2 -1814.017} C_VEL
LIN {X 0,Y 580.305,Z 487.199,A -85,B 0,C 180,E1 -1816.916,E2 -1816.916} C_VEL
LIN {X 0,Y 580.301,Z 487.196,A -85,B 0,C 180,E1 -1819.822,E2 -1819.822} C_VEL
LIN {X 0,Y 580.268,Z 487.199,A -85,B 0,C 180,E1 -1822.053,E2 -1822.053} C_VEL
LIN {X 0,Y 580.303,Z 487.204,A -85,B 0,C 180,E1 -1825.08,E2 -1825.08} C_VEL
LIN {X 0,Y 580.312,Z 487.193,A -85,B 0,C 180,E1 -1827.864,E2 -1827.864} C_VEL
LIN {X 0,Y 580.292,Z 487.199,A -85,B 0,C 180,E1 -1830.698,E2 -1830.698} C_VEL
LIN {X 0,Y 580.298,Z 487.2,A -85,B 0,C 180,E1 -1833.317,E2 -1833.317} C_VEL
LIN {X 0,Y 580.322,Z 487.192,A -85,B 0,C 180,E1 -1835.769,E2 -1835.769} C_VEL
LIN {X 0,Y 580.284,Z 487.196,A -85,B 0,C 180,E1 -1838.147,E2 -1838.147} C_VEL
LIN {X 0,Y 580.296,Z 487.203,A -85,B 0,C 180,E1 -1840.844,E2 -1840.844} C_VEL
LIN {X 0,Y 580.273,Z 487.199,A -85,B 0,C 180,E1 -1843.659,E2 -1843.659} C_VEL
LIN {X 0,Y 580.282,Z 487.202,A -85,B 0,C 180,E1 -1846.609,E2 -1846.609} C_VEL
LIN {X 0,Y 580.297,Z 487.202,A -85,B 0,C 180,E1 -1849.158,E2 -1849.158} C_VEL
LIN {X 0,Y 580.289,Z 487.196,A -85,B 0,C 180,E1 -1851.927,E2 -1851.927} C_VEL
LIN {X 0,Y 580.279,Z 487.201,A -85,B 0,C 180,E1 -1854.456,E2 -1854.456} C_VEL
LIN {X 0,Y 580.29,Z 487.206,A -85,B 0,C 180,E1 -1856.976,E2 -1856.976} C_VEL
LIN {X 0,Y 580.302,Z 487.198,A -85,B 0,C 180,E1 -1859.426,E2 -1859.426} C_VEL
LIN {X 0,Y 580.297,Z 487.197,A -85,B 0,C 180,E1 -1862.142,E2 -1862.142} C_VEL
LIN {X 0,Y 580.295,Z 487.251,A -85,B 0,C 180,E1 -1865.066,E2 -1865.066} C_VEL
LIN {X 0,Y 581.207,Z 491.898,A -85,B 0,C 180,E1 -1865.725,E2 -1865.725} C_VEL
LIN {X 0,Y 581.013,Z 513.568,A -85,B 0,C 180,E1 -1868.556,E2 -1868.556} C_VEL
LIN {X 0,Y 580.783,Z 537.818,A -85,B 0,C 180,E1 -1871.662,E2 -1871.662} C_VEL
LIN {X 0,Y 580.539,Z 562.213,A -85,B 0,C 180,E1 -1874.734,E2 -1874.734} C_VEL
LIN {X 0,Y 580.445,Z 574.948,A -85,B 0,C 180,E1 -1876.321,E2 -1876.321} C_VEL
LIN {X 0,Y 580.963,Z 579.746,A -85,B 0,C 180,E1 -1876.401,E2 -1876.401} C_VEL
LIN {X 0,Y 580.797,Z 683.961,A -85,B 0,C 180,E1 -1877.708,E2 -1877.708} C_VEL
LIN {X 0,Y 580.734,Z 697.224,A -85,B 0,C 180,E1 -1878.017,E2 -1878.017} C_VEL
LIN {X 0,Y 580.646,Z 710.153,A -85,B 0,C 180,E1 -1878.467,E2 -1878.467} C_VEL
LIN {X 0,Y 580.563,Z 721.636,A -85,B 0,C 180,E1 -1879.009,E2 -1879.009} C_VEL
LIN {X 0,Y 580.426,Z 733.206,A -85,B 0,C 180,E1 -1879.712,E2 -1879.712} C_VEL
LIN {X 0,Y 580.341,Z 743.601,A -85,B 0,C 180,E1 -1880.503,E2 -1880.503} C_VEL
LIN {X 0,Y 580.271,Z 752.115,A -85,B 0,C 180,E1 -1881.292,E2 -1881.292} C_VEL
LIN {X 0,Y 580.221,Z 759.962,A -85,B 0,C 180,E1 -1882.168,E2 -1882.168} C_VEL
LIN {X 0,Y 580.153,Z 767.651,A -85,B 0,C 180,E1 -1883.222,E2 -1883.222} C_VEL
LIN {X 0,Y 580.139,Z 774.681,A -85,B 0,C 180,E1 -1884.439,E2 -1884.439} C_VEL
LIN {X 0,Y 580.108,Z 779.372,A -85,B 0,C 180,E1 -1885.484,E2 -1885.484} C_VEL
LIN {X 0,Y 580.123,Z 782.958,A -85,B 0,C 180,E1 -1886.527,E2 -1886.527} C_VEL
LIN {X 0,Y 580.043,Z 784.81,A -85,B 0,C 180,E1 -1887.222,E2 -1887.222} C_VEL
LIN {X 0,Y 580.038,Z 786.201,A -85,B 0,C 180,E1 -1887.917,E2 -1887.917} C_VEL
LIN {X 0,Y 580.04,Z 787.785,A -85,B 0,C 180,E1 -1889.306,E2 -1889.306} C_VEL
LIN {X 0,Y 580.037,Z 788,A -85,B 0,C 180,E1 -1890,E2 -1890} C_VEL
LIN {X 0,Y 580.047,Z 787.185,A -85,B 0,C 180,E1 -1891.389,E2 -1891.389} C_VEL
LIN {X 0,Y 580.038,Z 786.2,A -85,B 0,C 180,E1 -1892.083,E2 -1892.083} C_VEL
LIN {X 0,Y 580.043,Z 784.809,A -85,B 0,C 180,E1 -1892.778,E2 -1892.778} C_VEL
LIN {X 0,Y 580.109,Z 781.896,A -85,B 0,C 180,E1 -1893.82,E2 -1893.82} C_VEL
LIN {X 0,Y 580.054,Z 777.95,A -85,B 0,C 180,E1 -1894.865,E2 -1894.865} C_VEL
LIN {X 0,Y 580.139,Z 771.878,A -85,B 0,C 180,E1 -1896.085,E2 -1896.085} C_VEL
LIN {X 0,Y 580.184,Z 765.238,A -85,B 0,C 180,E1 -1897.132,E2 -1897.132} C_VEL
LIN {X 0,Y 580.25,Z 756.992,A -85,B 0,C 180,E1 -1898.182,E2 -1898.182} C_VEL
LIN {X 0,Y 580.308,Z 748.54,A -85,B 0,C 180,E1 -1899.058,E2 -1899.058} C_VEL
LIN {X 0,Y 580.415,Z 738.099,A -85,B 0,C 180,E1 -1899.936,E2 -1899.936} C_VEL
LIN {X 0,Y 580.522,Z 727.76,A -85,B 0,C 180,E1 -1900.639,E2 -1900.639} C_VEL
LIN {X 0,Y 580.597,Z 716.238,A -85,B 0,C 180,E1 -1901.264,E2 -1901.264} C_VEL
LIN {X 0,Y 580.662,Z 703.484,A -85,B 0,C 180,E1 -1901.785,E2 -1901.785} C_VEL
LIN {X 0,Y 580.744,Z 690.451,A -85,B 0,C 180,E1 -1902.16,E2 -1902.16} C_VEL
LIN {X 0,Y 580.834,Z 678.106,A -85,B 0,C 180,E1 -1902.38,E2 -1902.38} C_VEL
LIN {X 0,Y 580.859,Z 577.956,A -85,B 0,C 180,E1 -1903.624,E2 -1903.624} C_VEL
LIN {X 0,Y 580.445,Z 574.948,A -85,B 0,C 180,E1 -1903.679,E2 -1903.679} C_VEL
LIN {X 0,Y 580.627,Z 552.168,A -85,B 0,C 180,E1 -1906.525,E2 -1906.525} C_VEL
LIN {X 0,Y 580.808,Z 530.312,A -85,B 0,C 180,E1 -1909.295,E2 -1909.295} C_VEL
LIN {X 0,Y 581.025,Z 509.118,A -85,B 0,C 180,E1 -1912.022,E2 -1912.022} C_VEL
LIN {X 0,Y 581.186,Z 491.898,A -85,B 0,C 180,E1 -1914.276,E2 -1914.276} C_VEL
LIN {X 0,Y 580.264,Z 487.209,A -85,B 0,C 180,E1 -1914.975,E2 -1914.975} C_VEL
LIN {X 0,Y 580.297,Z 487.197,A -85,B 0,C 180,E1 -1917.858,E2 -1917.858} C_VEL
LIN {X 0,Y 580.292,Z 487.199,A -85,B 0,C 180,E1 -1920.695,E2 -1920.695} C_VEL
LIN {X 0,Y 580.302,Z 487.203,A -85,B 0,C 180,E1 -1923.316,E2 -1923.316} C_VEL
LIN {X 0,Y 580.243,Z 487.203,A -85,B 0,C 180,E1 -1925.756,E2 -1925.756} C_VEL
LIN {X 0,Y 580.287,Z 487.192,A -85,B 0,C 180,E1 -1928.145,E2 -1928.145} C_VEL
LIN {X 0,Y 580.297,Z 487.199,A -85,B 0,C 180,E1 -1930.842,E2 -1930.842} C_VEL
LIN {X 0,Y 580.284,Z 487.199,A -85,B 0,C 180,E1 -1933.656,E2 -1933.656} C_VEL
LIN {X 0,Y 580.271,Z 487.2,A -85,B 0,C 180,E1 -1936.609,E2 -1936.609} C_VEL
LIN {X 0,Y 580.294,Z 487.204,A -85,B 0,C 180,E1 -1939.156,E2 -1939.156} C_VEL
LIN {X 0,Y 580.284,Z 487.197,A -85,B 0,C 180,E1 -1941.926,E2 -1941.926} C_VEL
LIN {X 0,Y 580.303,Z 487.194,A -85,B 0,C 180,E1 -1944.456,E2 -1944.456} C_VEL
LIN {X 0,Y 580.285,Z 487.204,A -85,B 0,C 180,E1 -1946.975,E2 -1946.975} C_VEL
LIN {X 0,Y 580.302,Z 487.199,A -85,B 0,C 180,E1 -1949.425,E2 -1949.425} C_VEL
LIN {X 0,Y 580.312,Z 487.193,A -85,B 0,C 180,E1 -1952.136,E2 -1952.136} C_VEL
LIN {X 0,Y 580.302,Z 487.2,A -85,B 0,C 180,E1 -1954.92,E2 -1954.92} C_VEL
LIN {X 0,Y 580.266,Z 487.198,A -85,B 0,C 180,E1 -1957.947,E2 -1957.947} C_VEL
LIN {X 0,Y 580.308,Z 487.2,A -85,B 0,C 180,E1 -1960.914,E2 -1960.914} C_VEL
LIN {X 0,Y 580.273,Z 487.196,A -85,B 0,C 180,E1 -1963.825,E2 -1963.825} C_VEL
LIN {X 0,Y 580.316,Z 487.192,A -85,B 0,C 180,E1 -1965.983,E2 -1965.983} C_VEL
LIN {X 0,Y 580.321,Z 487.197,A -85,B 0,C 180,E1 -1968.827,E2 -1968.827} C_VEL
LIN {X 0,Y 580.327,Z 487.191,A -85,B 0,C 180,E1 -1971.644,E2 -1971.644} C_VEL
LIN {X 0,Y 580.324,Z 487.192,A -85,B 0,C 180,E1 -1974.44,E2 -1974.44} C_VEL
LIN {X 0,Y 580.342,Z 487.197,A -85,B 0,C 180,E1 -1977.224,E2 -1977.224} C_VEL
LIN {X 0,Y 580.342,Z 487.186,A -85,B 0,C 180,E1 -1980,E2 -1980} C_VEL
LIN {X 0,Y 580.341,Z 487.193,A -85,B 0,C 180,E1 -1982.777,E2 -1982.777} C_VEL
LIN {X 0,Y 580.328,Z 487.193,A -85,B 0,C 180,E1 -1985.56,E2 -1985.56} C_VEL
LIN {X 0,Y 580.328,Z 487.189,A -85,B 0,C 180,E1 -1988.356,E2 -1988.356} C_VEL
LIN {X 0,Y 580.323,Z 487.2,A -85,B 0,C 180,E1 -1991.209,E2 -1991.209} C_VEL
LIN {X 0,Y 580.318,Z 487.192,A -85,B 0,C 180,E1 -1994.017,E2 -1994.017} C_VEL
LIN {X 0,Y 580.305,Z 487.199,A -85,B 0,C 180,E1 -1996.915,E2 -1996.915} C_VEL
LIN {X 0,Y 580.301,Z 487.195,A -85,B 0,C 180,E1 -1999.823,E2 -1999.823} C_VEL
LIN {X 0,Y 580.279,Z 487.202,A -85,B 0,C 180,E1 -2001.345,E2 -2001.345} C_VEL
LIN {X 0,Y 579.582,Z 487.285,A -85,B 0,C 180,E1 -2001.924,E2 -2001.924} C_VEL
LIN {X 0,Y 576.705,Z 487.648,A -85,B 0,C 180,E1 -2002.864,E2 -2002.864} C_VEL
LIN {X 0,Y 574.31,Z 487.942,A -85,B 0,C 180,E1 -2003.62,E2 -2003.62} C_VEL
LIN {X 0,Y 573.311,Z 488.064,A -85,B 0,C 180,E1 -2004.204,E2 -2004.204} C_VEL
LIN {X 0,Y 573.244,Z 488.073,A -85,B 0,C 180,E1 -2004.401,E2 -2004.401} C_VEL
LIN {X 0,Y 573.262,Z 488.08,A -85,B 0,C 180,E1 -2006.976,E2 -2006.976} C_VEL
LIN {X 0,Y 573.249,Z 488.075,A -85,B 0,C 180,E1 -2009.491,E2 -2009.491} C_VEL
LIN {X 0,Y 573.25,Z 488.073,A -85,B 0,C 180,E1 -2012.23,E2 -2012.23} C_VEL
LIN {X 0,Y 573.249,Z 488.078,A -85,B 0,C 180,E1 -2014.775,E2 -2014.775} C_VEL
LIN {X 0,Y 573.251,Z 488.081,A -85,B 0,C 180,E1 -2017.167,E2 -2017.167} C_VEL
LIN {X 0,Y 573.246,Z 488.075,A -85,B 0,C 180,E1 -2019.608,E2 -2019.608} C_VEL
LIN {X 0,Y 573.24,Z 488.079,A -85,B 0,C 180,E1 -2022.643,E2 -2022.643} C_VEL
